LIN {X 0,Y 573.115,Z 294.058,A -85,B 0,C 180,E1 -2039.137,E2 -2039.137} C_VEL
LIN {X 0,Y 573.081,Z 298.172,A -85,B 0,C 180,E1 -2042.003,E2 -2042.003} C_VEL
LIN {X 0,Y 573.022,Z 301.873,A -85,B 0,C 180,E1 -2044.579,E2 -2044.579} C_VEL
LIN {X 0,Y 573.043,Z 305.517,A -85,B 0,C 180,E1 -2046.901,E2 -2046.901} C_VEL
LIN {X 0,Y 572.998,Z 309.134,A -85,B 0,C 180,E1 -2049.164,E2 -2049.164} C_VEL
LIN {X 0,Y 573.01,Z 312.764,A -85,B 0,C 180,E1 -2051.404,E2 -2051.404} C_VEL
LIN {X 0,Y 572.982,Z 314.48,A -85,B 0,C 180,E1 -2052.451,E2 -2052.451} C_VEL
LIN {X 0,Y 574.741,Z 322.312,A -85,B 0,C 180,E1 -2052.634,E2 -2052.634} C_VEL
LIN {X 0,Y 574.641,Z 337.953,A -85,B 0,C 180,E1 -2052.982,E2 -2052.982} C_VEL
LIN {X 0,Y 574.406,Z 353.082,A -85,B 0,C 180,E1 -2053.478,E2 -2053.478} C_VEL
LIN {X 0,Y 574.266,Z 365.728,A -85,B 0,C 180,E1 -2054.016,E2 -2054.016} C_VEL
LIN {X 0,Y 574.068,Z 377.863,A -85,B 0,C 180,E1 -2054.648,E2 -2054.648} C_VEL
LIN {X 0,Y 573.885,Z 391.295,A -85,B 0,C 180,E1 -2055.496,E2 -2055.496} C_VEL
LIN {X 0,Y 573.651,Z 404.761,A -85,B 0,C 180,E1 -2056.539,E2 -2056.539} C_VEL
LIN {X 0,Y 573.479,Z 416.274,A -85,B 0,C 180,E1 -2057.616,E2 -2057.616} C_VEL
LIN {X 0,Y 573.311,Z 426.306,A -85,B 0,C 180,E1 -2058.722,E2 -2058.722} C_VEL
LIN {X 0,Y 573.203,Z 436.788,A -85,B 0,C 180,E1 -2060.116,E2 -2060.116} C_VEL
LIN {X 0,Y 573.134,Z 444.469,A -85,B 0,C 180,E1 -2061.36,E2 -2061.36} C_VEL
LIN {X 0,Y 573.076,Z 450.883,A -85,B 0,C 180,E1 -2062.601,E2 -2062.601} C_VEL
LIN {X 0,Y 573.042,Z 456.782,A -85,B 0,C 180,E1 -2064.016,E2 -2064.016} C_VEL
LIN {X 0,Y 572.949,Z 460.255,A -85,B 0,C 180,E1 -2065.074,E2 -2065.074} C_VEL
LIN {X 0,Y 573.004,Z 463.808,A -85,B 0,C 180,E1 -2066.484,E2 -2066.484} C_VEL
LIN {X 0,Y 572.938,Z 466.135,A -85,B 0,C 180,E1 -2067.891,E2 -2067.891} C_VEL
LIN {X 0,Y 572.936,Z 467.306,A -85,B 0,C 180,E1 -2069.297,E2 -2069.297} C_VEL
LIN {X 0,Y 572.937,Z 467.337,A -85,B 0,C 180,E1 -2070.703,E2 -2070.703} C_VEL
LIN {X 0,Y 572.939,Z 466.235,A -85,B 0,C 180,E1 -2072.109,E2 -2072.109} C_VEL
LIN {X 0,Y 573.006,Z 463.992,A -85,B 0,C 180,E1 -2073.516,E2 -2073.516} C_VEL
LIN {X 0,Y 572.949,Z 460.527,A -85,B 0,C 180,E1 -2074.926,E2 -2074.926} C_VEL
LIN {X 0,Y 573.042,Z 457.098,A -85,B 0,C 180,E1 -2075.984,E2 -2075.984} C_VEL
LIN {X 0,Y 573.071,Z 451.302,A -85,B 0,C 180,E1 -2077.398,E2 -2077.398} C_VEL
LIN {X 0,Y 573.132,Z 444.977,A -85,B 0,C 180,E1 -2078.639,E2 -2078.639} C_VEL
LIN {X 0,Y 573.2,Z 437.38,A -85,B 0,C 180,E1 -2079.884,E2 -2079.884} C_VEL
LIN {X 0,Y 573.287,Z 428.365,A -85,B 0,C 180,E1 -2081.119,E2 -2081.119} C_VEL
LIN {X 0,Y 573.464,Z 417.166,A -85,B 0,C 180,E1 -2082.384,E2 -2082.384} C_VEL
LIN {X 0,Y 573.644,Z 406.815,A -85,B 0,C 180,E1 -2083.37,E2 -2083.37} C_VEL
LIN {X 0,Y 573.838,Z 395.714,A -85,B 0,C 180,E1 -2084.27,E2 -2084.27} C_VEL
LIN {X 0,Y 574.004,Z 382.508,A -85,B 0,C 180,E1 -2085.172,E2 -2085.172} C_VEL
LIN {X 0,Y 574.232,Z 369.513,A -85,B 0,C 180,E1 -2085.893,E2 -2085.893} C_VEL
LIN {X 0,Y 574.375,Z 356.387,A -85,B 0,C 180,E1 -2086.482,E2 -2086.482} C_VEL
LIN {X 0,Y 574.554,Z 342.236,A -85,B 0,C 180,E1 -2086.98,E2 -2086.98} C_VEL
LIN {X 0,Y 574.717,Z 327.066,A -85,B 0,C 180,E1 -2087.368,E2 -2087.368} C_VEL
LIN {X 0,Y 574.563,Z 321.22,A -85,B 0,C 180,E1 -2087.48,E2 -2087.48} C_VEL
LIN {X 0,Y 572.988,Z 314.455,A -85,B 0,C 180,E1 -2087.654,E2 -2087.654} C_VEL
LIN {X 0,Y 572.994,Z 310.49,A -85,B 0,C 180,E1 -2090.086,E2 -2090.086} C_VEL
LIN {X 0,Y 573.008,Z 306.857,A -85,B 0,C 180,E1 -2092.347,E2 -2092.347} C_VEL
LIN {X 0,Y 573.025,Z 302.942,A -85,B 0,C 180,E1 -2094.825,E2 -2094.825} C_VEL
LIN {X 0,Y 573.07,Z 299.762,A -85,B 0,C 180,E1 -2096.985,E2 -2096.985} C_VEL
LIN {X 0,Y 573.105,Z 296.219,A -85,B 0,C 180,E1 -2099.463,E2 -2099.463} C_VEL
LIN {X 0,Y 573.144,Z 292.244,A -85,B 0,C 180,E1 -2102.211,E2 -2102.211} C_VEL
LIN {X 0,Y 573.162,Z 287.996,A -85,B 0,C 180,E1 -2105.191,E2 -2105.191} C_VEL
LIN {X 0,Y 573.212,Z 284.101,A -85,B 0,C 180,E1 -2107.809,E2 -2107.809} C_VEL
LIN {X 0,Y 573.201,Z 279.714,A -85,B 0,C 180,E1 -2110.529,E2 -2110.529} C_VEL
LIN {X 0,Y 573.239,Z 279.706,A -85,B 0,C 180,E1 -2113.359,E2 -2113.359} C_VEL
LIN {X 0,Y 573.24,Z 279.703,A -85,B 0,C 180,E1 -2116.332,E2 -2116.332} C_VEL
LIN {X 0,Y 573.228,Z 279.71,A -85,B 0,C 180,E1 -2118.543,E2 -2118.543} C_VEL
LIN {X 0,Y 573.23,Z 279.703,A -85,B 0,C 180,E1 -2121.297,E2 -2121.297} C_VEL
LIN {X 0,Y 573.22,Z 279.707,A -85,B 0,C 180,E1 -2124.018,E2 -2124.018} C_VEL
LIN {X 0,Y 573.27,Z 279.7,A -85,B 0,C 180,E1 -2126.518,E2 -2126.518} C_VEL
LIN {X 0,Y 573.226,Z 279.704,A -85,B 0,C 180,E1 -2129.118,E2 -2129.118} C_VEL
LIN {X 0,Y 573.194,Z 279.714,A -85,B 0,C 180,E1 -2131.982,E2 -2131.982} C_VEL
LIN {X 0,Y 573.238,Z 279.701,A -85,B 0,C 180,E1 -2134.589,E2 -2134.589} C_VEL
LIN {X 0,Y 573.236,Z 279.701,A -85,B 0,C 180,E1 -2137.662,E2 -2137.662} C_VEL
LIN {X 0,Y 573.267,Z 279.701,A -85,B 0,C 180,E1 -2140.67,E2 -2140.67} C_VEL
LIN {X 0,Y 573.221,Z 279.709,A -85,B 0,C 180,E1 -2143.621,E2 -2143.621} C_VEL
LIN {X 0,Y 573.273,Z 279.699,A -85,B 0,C 180,E1 -2145.807,E2 -2145.807} C_VEL
LIN {X 0,Y 573.264,Z 279.703,A -85,B 0,C 180,E1 -2148.745,E2 -2148.745} C_VEL
LIN {X 0,Y 573.252,Z 279.703,A -85,B 0,C 180,E1 -2151.54,E2 -2151.54} C_VEL
LIN {X 0,Y 573.262,Z 279.697,A -85,B 0,C 180,E1 -2154.371,E2 -2154.371} C_VEL
LIN {X 0,Y 573.309,Z 279.697,A -85,B 0,C 180,E1 -2157.189,E2 -2157.189} C_VEL
LIN {X 0,Y 573.324,Z 279.693,A -85,B 0,C 180,E1 -2160,E2 -2160} C_VEL
LIN {X 0,Y 573.287,Z 279.696,A -85,B 0,C 180,E1 -2162.811,E2 -2162.811} C_VEL
LIN {X 0,Y 573.28,Z 279.698,A -85,B 0,C 180,E1 -2165.628,E2 -2165.628} C_VEL
LIN {X 0,Y 573.255,Z 279.706,A -85,B 0,C 180,E1 -2168.46,E2 -2168.46} C_VEL
LIN {X 0,Y 573.273,Z 279.696,A -85,B 0,C 180,E1 -2171.312,E2 -2171.312} C_VEL
LIN {X 0,Y 573.244,Z 279.701,A -85,B 0,C 180,E1 -2174.409,E2 -2174.409} C_VEL
LIN {X 0,Y 573.247,Z 279.705,A -85,B 0,C 180,E1 -2177.112,E2 -2177.112} C_VEL
LIN {X 0,Y 573.253,Z 279.705,A -85,B 0,C 180,E1 -2180.077,E2 -2180.077} C_VEL
LIN {X 0,Y 573.235,Z 279.703,A -85,B 0,C 180,E1 -2183.099,E2 -2183.099} C_VEL
LIN {X 0,Y 573.233,Z 279.702,A -85,B 0,C 180,E1 -2186.191,E2 -2186.191} C_VEL
LIN {X 0,Y 573.229,Z 279.71,A -85,B 0,C 180,E1 -2188.565,E2 -2188.565} C_VEL
LIN {X 0,Y 573.23,Z 279.703,A -85,B 0,C 180,E1 -2190.993,E2 -2190.993} C_VEL
LIN {X 0,Y 573.263,Z 279.706,A -85,B 0,C 180,E1 -2193.524,E2 -2193.524} C_VEL
LIN {X 0,Y 573.19,Z 279.708,A -85,B 0,C 180,E1 -2196.053,E2 -2196.053} C_VEL
LIN {X 0,Y 573.232,Z 279.708,A -85,B 0,C 180,E1 -2198.702,E2 -2198.702} C_VEL
LIN {X 0,Y 573.237,Z 279.706,A -85,B 0,C 180,E1 -2201.594,E2 -2201.594} C_VEL
LIN {X 0,Y 573.225,Z 279.703,A -85,B 0,C 180,E1 -2204.334,E2 -2204.334} C_VEL
LIN {X 0,Y 573.218,Z 279.706,A -85,B 0,C 180,E1 -2207.361,E2 -2207.361} C_VEL
LIN {X 0,Y 573.236,Z 279.709,A -85,B 0,C 180,E1 -2210.392,E2 -2210.392} C_VEL
LIN {X 0,Y 573.252,Z 279.707,A -85,B 0,C 180,E1 -2213.078,E2 -2213.078} C_VEL
LIN {X 0,Y 573.217,Z 279.814,A -85,B 0,C 180,E1 -2214.166,E2 -2214.166} C_VEL
LIN {X 0,Y 575.333,Z 288.451,A -85,B 0,C 180,E1 -2215.812,E2 -2215.812} C_VEL
LIN {X 0,Y 574.902,Z 304.368,A -85,B 0,C 180,E1 -2218.459,E2 -2218.459} C_VEL
LIN {X 0,Y 574.675,Z 320.037,A -85,B 0,C 180,E1 -2220.914,E2 -2220.914} C_VEL
LIN {X 0,Y 574.403,Z 337.41,A -85,B 0,C 180,E1 -2223.567,E2 -2223.567} C_VEL
LIN {X 0,Y 574.164,Z 354.72,A -85,B 0,C 180,E1 -2226.176,E2 -2226.176} C_VEL
LIN {X 0,Y 573.88,Z 375.193,A -85,B 0,C 180,E1 -2229.198,E2 -2229.198} C_VEL
LIN {X 0,Y 573.658,Z 394.386,A -85,B 0,C 180,E1 -2231.98,E2 -2231.98} C_VEL
LIN {X 0,Y 573.656,Z 396.802,A -85,B 0,C 180,E1 -2232.329,E2 -2232.329} C_VEL
LIN {X 0,Y 574.768,Z 403.436,A -85,B 0,C 180,E1 -2232.451,E2 -2232.451} C_VEL
LIN {X 0,Y 574.667,Z 419.595,A -85,B 0,C 180,E1 -2232.729,E2 -2232.729} C_VEL
LIN {X 0,Y 574.555,Z 435.297,A -85,B 0,C 180,E1 -2233.157,E2 -2233.157} C_VEL
LIN {X 0,Y 574.348,Z 449.799,A -85,B 0,C 180,E1 -2233.7,E2 -2233.7} C_VEL
LIN {X 0,Y 574.157,Z 463.874,A -85,B 0,C 180,E1 -2234.378,E2 -2234.378} C_VEL
LIN {X 0,Y 573.982,Z 476.044,A -85,B 0,C 180,E1 -2235.1,E2 -2235.1} C_VEL
LIN {X 0,Y 573.748,Z 488.699,A -85,B 0,C 180,E1 -2236,E2 -2236} C_VEL
LIN {X 0,Y 573.581,Z 499.336,A -85,B 0,C 180,E1 -2236.899,E2 -2236.899} C_VEL
LIN {X 0,Y 573.405,Z 510.141,A -85,B 0,C 180,E1 -2237.974,E2 -2237.974} C_VEL
LIN {X 0,Y 573.3,Z 519.79,A -85,B 0,C 180,E1 -2239.111,E2 -2239.111} C_VEL
LIN {X 0,Y 573.188,Z 528.295,A -85,B 0,C 180,E1 -2240.294,E2 -2240.294} C_VEL
LIN {X 0,Y 573.109,Z 535.751,A -85,B 0,C 180,E1 -2241.538,E2 -2241.538} C_VEL
LIN {X 0,Y 573.047,Z 542.702,A -85,B 0,C 180,E1 -2242.956,E2 -2242.956} C_VEL
LIN {X 0,Y 573.055,Z 548.161,A -85,B 0,C 180,E1 -2244.37,E2 -2244.37} C_VEL
LIN {X 0,Y 573.006,Z 552.29,A -85,B 0,C 180,E1 -2245.78,E2 -2245.78} C_VEL
LIN {X 0,Y 572.955,Z 555.188,A -85,B 0,C 180,E1 -2247.188,E2 -2247.188} C_VEL
LIN {X 0,Y 572.944,Z 556.912,A -85,B 0,C 180,E1 -2248.594,E2 -2248.594} C_VEL
LIN {X 0,Y 572.935,Z 557.5,A -85,B 0,C 180,E1 -2250,E2 -2250} C_VEL
LIN {X 0,Y 572.944,Z 556.911,A -85,B 0,C 180,E1 -2251.406,E2 -2251.406} C_VEL
LIN {X 0,Y 572.955,Z 555.186,A -85,B 0,C 180,E1 -2252.813,E2 -2252.813} C_VEL
LIN {X 0,Y 573.007,Z 552.288,A -85,B 0,C 180,E1 -2254.22,E2 -2254.22} C_VEL
LIN {X 0,Y 573.055,Z 548.162,A -85,B 0,C 180,E1 -2255.631,E2 -2255.631} C_VEL
LIN {X 0,Y 573.048,Z 542.701,A -85,B 0,C 180,E1 -2257.045,E2 -2257.045} C_VEL
LIN {X 0,Y 573.109,Z 535.748,A -85,B 0,C 180,E1 -2258.462,E2 -2258.462} C_VEL
LIN {X 0,Y 573.199,Z 527.087,A -85,B 0,C 180,E1 -2259.884,E2 -2259.884} C_VEL
LIN {X 0,Y 573.295,Z 517.948,A -85,B 0,C 180,E1 -2261.124,E2 -2261.124} C_VEL
LIN {X 0,Y 573.453,Z 508.507,A -85,B 0,C 180,E1 -2262.205,E2 -2262.205} C_VEL
LIN {X 0,Y 573.628,Z 497.383,A -85,B 0,C 180,E1 -2263.281,E2 -2263.281} C_VEL
LIN {X 0,Y 573.828,Z 485.135,A -85,B 0,C 180,E1 -2264.274,E2 -2264.274} C_VEL
LIN {X 0,Y 574.016,Z 471.775,A -85,B 0,C 180,E1 -2265.172,E2 -2265.172} C_VEL
LIN {X 0,Y 574.222,Z 458.597,A -85,B 0,C 180,E1 -2265.894,E2 -2265.894} C_VEL
LIN {X 0,Y 574.416,Z 444.173,A -85,B 0,C 180,E1 -2266.527,E2 -2266.527} C_VEL
LIN {X 0,Y 574.592,Z 429.245,A -85,B 0,C 180,E1 -2267.025,E2 -2267.025} C_VEL
LIN {X 0,Y 574.68,Z 414.321,A -85,B 0,C 180,E1 -2267.377,E2 -2267.377} C_VEL
LIN {X 0,Y 574.609,Z 401.989,A -85,B 0,C 180,E1 -2267.572,E2 -2267.572} C_VEL
LIN {X 0,Y 573.643,Z 396.706,A -85,B 0,C 180,E1 -2267.686,E2 -2267.686} C_VEL
LIN {X 0,Y 573.874,Z 377.749,A -85,B 0,C 180,E1 -2270.428,E2 -2270.428} C_VEL
LIN {X 0,Y 574.128,Z 357.888,A -85,B 0,C 180,E1 -2273.352,E2 -2273.352} C_VEL
LIN {X 0,Y 574.401,Z 339.363,A -85,B 0,C 180,E1 -2276.134,E2 -2276.134} C_VEL
LIN {X 0,Y 574.615,Z 323.851,A -85,B 0,C 180,E1 -2278.49,E2 -2278.49} C_VEL
LIN {X 0,Y 574.762,Z 310.765,A -85,B 0,C 180,E1 -2280.494,E2 -2280.494} C_VEL
LIN {X 0,Y 575.281,Z 296.37,A -85,B 0,C 180,E1 -2282.932,E2 -2282.932} C_VEL
LIN {X 0,Y 575.707,Z 289.67,A -85,B 0,C 180,E1 -2284.163,E2 -2284.163} C_VEL
LIN {X 0,Y 574.296,Z 283.704,A -85,B 0,C 180,E1 -2285.541,E2 -2285.541} C_VEL
LIN {X 0,Y 573.22,Z 279.71,A -85,B 0,C 180,E1 -2286.651,E2 -2286.651} C_VEL
LIN {X 0,Y 573.247,Z 279.707,A -85,B 0,C 180,E1 -2289.607,E2 -2289.607} C_VEL
LIN {X 0,Y 573.245,Z 279.708,A -85,B 0,C 180,E1 -2292.642,E2 -2292.642} C_VEL
LIN {X 0,Y 573.224,Z 279.709,A -85,B 0,C 180,E1 -2295.665,E2 -2295.665} C_VEL
LIN {X 0,Y 573.234,Z 279.707,A -85,B 0,C 180,E1 -2298.543,E2 -2298.543} C_VEL
LIN {X 0,Y 573.245,Z 279.706,A -85,B 0,C 180,E1 -2301.299,E2 -2301.299} C_VEL
LIN {X 0,Y 573.189,Z 279.715,A -85,B 0,C 180,E1 -2304.022,E2 -2304.022} C_VEL
LIN {X 0,Y 573.289,Z 282.484,A -85,B 0,C 180,E1 -2306.519,E2 -2306.519} C_VEL
LIN {X 0,Y 573.241,Z 285.279,A -85,B 0,C 180,E1 -2309.116,E2 -2309.116} C_VEL
LIN {X 0,Y 573.262,Z 287.554,A -85,B 0,C 180,E1 -2311.437,E2 -2311.437} C_VEL
LIN {X 0,Y 573.201,Z 289.676,A -85,B 0,C 180,E1 -2313.807,E2 -2313.807} C_VEL
LIN {X 0,Y 573.084,Z 291.517,A -85,B 0,C 180,E1 -2316.128,E2 -2316.128} C_VEL
LIN {X 0,Y 572.988,Z 294.122,A -85,B 0,C 180,E1 -2319.164,E2 -2319.164} C_VEL
LIN {X 0,Y 572.965,Z 296.701,A -85,B 0,C 180,E1 -2321.403,E2 -2321.403} C_VEL
LIN {X 0,Y 572.967,Z 299.405,A -85,B 0,C 180,E1 -2323.613,E2 -2323.613} C_VEL
LIN {X 0,Y 572.986,Z 303.009,A -85,B 0,C 180,E1 -2326.524,E2 -2326.524} C_VEL
LIN {X 0,Y 572.999,Z 304.333,A -85,B 0,C 180,E1 -2327.583,E2 -2327.583} C_VEL
LIN {X 0,Y 573.818,Z 310.855,A -85,B 0,C 180,E1 -2327.758,E2 -2327.758} C_VEL
LIN {X 0,Y 573.71,Z 324.273,A -85,B 0,C 180,E1 -2328.16,E2 -2328.16} C_VEL
LIN {X 0,Y 573.629,Z 336.787,A -85,B 0,C 180,E1 -2328.695,E2 -2328.695} C_VEL
LIN {X 0,Y 573.528,Z 347.998,A -85,B 0,C 180,E1 -2329.321,E2 -2329.321} C_VEL
LIN {X 0,Y 573.35,Z 359.337,A -85,B 0,C 180,E1 -2330.119,E2 -2330.119} C_VEL
LIN {X 0,Y 573.28,Z 369.385,A -85,B 0,C 180,E1 -2331.008,E2 -2331.008} C_VEL
LIN {X 0,Y 573.161,Z 379.087,A -85,B 0,C 180,E1 -2332.071,E2 -2332.071} C_VEL
LIN {X 0,Y 573.093,Z 387.022,A -85,B 0,C 180,E1 -2333.163,E2 -2333.163} C_VEL
LIN {X 0,Y 573.07,Z 393.948,A -85,B 0,C 180,E1 -2334.37,E2 -2334.37} C_VEL
LIN {X 0,Y 573.029,Z 398.691,A -85,B 0,C 180,E1 -2335.428,E2 -2335.428} C_VEL
LIN {X 0,Y 573.023,Z 402.323,A -85,B 0,C 180,E1 -2336.484,E2 -2336.484} C_VEL
LIN {X 0,Y 572.959,Z 404.2,A -85,B 0,C 180,E1 -2337.188,E2 -2337.188} C_VEL
LIN {X 0,Y 572.938,Z 405.627,A -85,B 0,C 180,E1 -2337.891,E2 -2337.891} C_VEL
LIN {X 0,Y 572.942,Z 407.255,A -85,B 0,C 180,E1 -2339.297,E2 -2339.297} C_VEL
LIN {X 0,Y 572.938,Z 407.496,A -85,B 0,C 180,E1 -2340,E2 -2340} C_VEL
LIN {X 0,Y 572.941,Z 407.315,A -85,B 0,C 180,E1 -2340.703,E2 -2340.703} C_VEL
LIN {X 0,Y 572.937,Z 405.772,A -85,B 0,C 180,E1 -2342.109,E2 -2342.109} C_VEL
LIN {X 0,Y 572.96,Z 404.411,A -85,B 0,C 180,E1 -2342.812,E2 -2342.812} C_VEL
LIN {X 0,Y 573.015,Z 401.532,A -85,B 0,C 180,E1 -2343.868,E2 -2343.868} C_VEL
LIN {X 0,Y 572.963,Z 397.631,A -85,B 0,C 180,E1 -2344.926,E2 -2344.926} C_VEL
LIN {X 0,Y 573.075,Z 392.601,A -85,B 0,C 180,E1 -2345.984,E2 -2345.984} C_VEL
LIN {X 0,Y 573.083,Z 386.275,A -85,B 0,C 180,E1 -2347.044,E2 -2347.044} C_VEL
LIN {X 0,Y 573.175,Z 378.354,A -85,B 0,C 180,E1 -2348.106,E2 -2348.106} C_VEL
LIN {X 0,Y 573.287,Z 368.504,A -85,B 0,C 180,E1 -2349.17,E2 -2349.17} C_VEL
LIN {X 0,Y 573.416,Z 358.18,A -85,B 0,C 180,E1 -2350.059,E2 -2350.059} C_VEL
LIN {X 0,Y 573.544,Z 346.593,A -85,B 0,C 180,E1 -2350.856,E2 -2350.856} C_VEL
LIN {X 0,Y 573.658,Z 335.698,A -85,B 0,C 180,E1 -2351.449,E2 -2351.449} C_VEL
LIN {X 0,Y 573.718,Z 324.526,A -85,B 0,C 180,E1 -2351.921,E2 -2351.921} C_VEL
LIN {X 0,Y 573.827,Z 311.765,A -85,B 0,C 180,E1 -2352.309,E2 -2352.309} C_VEL
LIN {X 0,Y 573.379,Z 307.024,A -85,B 0,C 180,E1 -2352.428,E2 -2352.428} C_VEL
LIN {X 0,Y 572.963,Z 304.333,A -85,B 0,C 180,E1 -2352.508,E2 -2352.508} C_VEL
LIN {X 0,Y 572.959,Z 301.318,A -85,B 0,C 180,E1 -2354.927,E2 -2354.927} C_VEL
LIN {X 0,Y 572.943,Z 298.246,A -85,B 0,C 180,E1 -2357.422,E2 -2357.422} C_VEL
LIN {X 0,Y 572.979,Z 295.007,A -85,B 0,C 180,E1 -2360.087,E2 -2360.087} C_VEL
LIN {X 0,Y 572.968,Z 294.558,A -85,B 0,C 180,E1 -2360.463,E2 -2360.463} C_VEL
LIN {X 0,Y 572.312,Z 293.943,A -85,B 0,C 180,E1 -2361.046,E2 -2361.046} C_VEL
LIN {X 0,Y 569.466,Z 293.15,A -85,B 0,C 180,E1 -2361.995,E2 -2361.995} C_VEL
LIN {X 0,Y 567.052,Z 292.543,A -85,B 0,C 180,E1 -2362.759,E2 -2362.759} C_VEL
LIN {X 0,Y 566.01,Z 292.015,A -85,B 0,C 180,E1 -2363.348,E2 -2363.348} C_VEL
LIN {X 0,Y 565.923,Z 291.817,A -85,B 0,C 180,E1 -2363.547,E2 -2363.547} C_VEL
LIN {X 0,Y 565.974,Z 289.57,A -85,B 0,C 180,E1 -2365.761,E2 -2365.761} C_VEL
LIN {X 0,Y 566.002,Z 286.959,A -85,B 0,C 180,E1 -2368.163,E2 -2368.163} C_VEL
LIN {X 0,Y 565.98,Z 284.379,A -85,B 0,C 180,E1 -2370.605,E2 -2370.605} C_VEL
LIN {X 0,Y 565.98,Z 281.51,A -85,B 0,C 180,E1 -2373.118,E2 -2373.118} C_VEL
LIN {X 0,Y 566.008,Z 280.61,A -85,B 0,C 180,E1 -2373.97,E2 -2373.97} C_VEL
LIN {X 0,Y 566.194,Z 280.58,A -85,B 0,C 180,E1 -2376.57,E2 -2376.57} C_VEL
LIN {X 0,Y 566.225,Z 280.575,A -85,B 0,C 180,E1 -2379.687,E2 -2379.687} C_VEL
LIN {X 0,Y 566.203,Z 280.58,A -85,B 0,C 180,E1 -2382.917,E2 -2382.917} C_VEL
LIN {X 0,Y 566.161,Z 280.588,A -85,B 0,C 180,E1 -2385.96,E2 -2385.96} C_VEL
LIN {X 0,Y 566.168,Z 280.589,A -85,B 0,C 180,E1 -2388.142,E2 -2388.142} C_VEL
LIN {X 0,Y 566.136,Z 280.74,A -85,B 0,C 180,E1 -2389.794,E2 -2389.794} C_VEL
LIN {X 0,Y 566.165,Z 285.409,A -85,B 0,C 180,E1 -2392.604,E2 -2392.604} C_VEL
LIN {X 0,Y 566.113,Z 289.214,A -85,B 0,C 180,E1 -2395.175,E2 -2395.175} C_VEL
LIN {X 0,Y 566.091,Z 292.826,A -85,B 0,C 180,E1 -2397.734,E2 -2397.734} C_VEL
LIN {X 0,Y 566.052,Z 296.586,A -85,B 0,C 180,E1 -2400.355,E2 -2400.355} C_VEL
LIN {X 0,Y 566.001,Z 299.877,A -85,B 0,C 180,E1 -2402.65,E2 -2402.65} C_VEL
LIN {X 0,Y 565.963,Z 303.211,A -85,B 0,C 180,E1 -2405.026,E2 -2405.026} C_VEL
LIN {X 0,Y 565.948,Z 306.714,A -85,B 0,C 180,E1 -2407.358,E2 -2407.358} C_VEL
LIN {X 0,Y 565.931,Z 311.555,A -85,B 0,C 180,E1 -2410.409,E2 -2410.409} C_VEL
LIN {X 0,Y 565.893,Z 314.463,A -85,B 0,C 180,E1 -2412.213,E2 -2412.213} C_VEL
LIN {X 0,Y 567.959,Z 323.511,A -85,B 0,C 180,E1 -2412.44,E2 -2412.44} C_VEL
LIN {X 0,Y 567.805,Z 340.105,A -85,B 0,C 180,E1 -2412.836,E2 -2412.836} C_VEL
LIN {X 0,Y 567.57,Z 353.381,A -85,B 0,C 180,E1 -2413.285,E2 -2413.285} C_VEL
LIN {X 0,Y 567.408,Z 365.723,A -85,B 0,C 180,E1 -2413.818,E2 -2413.818} C_VEL
LIN {X 0,Y 567.203,Z 377.86,A -85,B 0,C 180,E1 -2414.458,E2 -2414.458} C_VEL
LIN {X 0,Y 567,Z 390.624,A -85,B 0,C 180,E1 -2415.268,E2 -2415.268} C_VEL
LIN {X 0,Y 566.727,Z 403.712,A -85,B 0,C 180,E1 -2416.28,E2 -2416.28} C_VEL
LIN {X 0,Y 566.535,Z 414.488,A -85,B 0,C 180,E1 -2417.279,E2 -2417.279} C_VEL
LIN {X 0,Y 566.338,Z 424.498,A -85,B 0,C 180,E1 -2418.366,E2 -2418.366} C_VEL
LIN {X 0,Y 566.226,Z 434.328,A -85,B 0,C 180,E1 -2419.632,E2 -2419.632} C_VEL
LIN {X 0,Y 566.057,Z 443.461,A -85,B 0,C 180,E1 -2421.072,E2 -2421.072} C_VEL
LIN {X 0,Y 566.016,Z 449.187,A -85,B 0,C 180,E1 -2422.15,E2 -2422.15} C_VEL
LIN {X 0,Y 565.946,Z 454.844,A -85,B 0,C 180,E1 -2423.44,E2 -2423.44} C_VEL
LIN {X 0,Y 565.926,Z 459.16,A -85,B 0,C 180,E1 -2424.656,E2 -2424.656} C_VEL
LIN {X 0,Y 565.913,Z 462.163,A -85,B 0,C 180,E1 -2425.727,E2 -2425.727} C_VEL
LIN {X 0,Y 565.872,Z 465.109,A -85,B 0,C 180,E1 -2427.152,E2 -2427.152} C_VEL
LIN {X 0,Y 565.842,Z 466.88,A -85,B 0,C 180,E1 -2428.576,E2 -2428.576} C_VEL
LIN {X 0,Y 565.837,Z 467.496,A -85,B 0,C 180,E1 -2430,E2 -2430} C_VEL
LIN {X 0,Y 565.844,Z 466.959,A -85,B 0,C 180,E1 -2431.423,E2 -2431.423} C_VEL
LIN {X 0,Y 565.874,Z 465.262,A -85,B 0,C 180,E1 -2432.847,E2 -2432.847} C_VEL
LIN {X 0,Y 565.913,Z 462.382,A -85,B 0,C 180,E1 -2434.273,E2 -2434.273} C_VEL
LIN {X 0,Y 565.982,Z 458.318,A -85,B 0,C 180,E1 -2435.701,E2 -2435.701} C_VEL
LIN {X 0,Y 565.974,Z 452.914,A -85,B 0,C 180,E1 -2437.133,E2 -2437.133} C_VEL
LIN {X 0,Y 566.058,Z 445.968,A -85,B 0,C 180,E1 -2438.568,E2 -2438.568} C_VEL
LIN {X 0,Y 566.125,Z 438.535,A -85,B 0,C 180,E1 -2439.828,E2 -2439.828} C_VEL
LIN {X 0,Y 566.253,Z 430.628,A -85,B 0,C 180,E1 -2440.956,E2 -2440.956} C_VEL
LIN {X 0,Y 566.415,Z 420.564,A -85,B 0,C 180,E1 -2442.177,E2 -2442.177} C_VEL
LIN {X 0,Y 566.627,Z 408.849,A -85,B 0,C 180,E1 -2443.356,E2 -2443.356} C_VEL
LIN {X 0,Y 566.833,Z 398.076,A -85,B 0,C 180,E1 -2444.266,E2 -2444.266} C_VEL
LIN {X 0,Y 567.092,Z 386.68,A -85,B 0,C 180,E1 -2445.085,E2 -2445.085} C_VEL
LIN {X 0,Y 567.267,Z 374.623,A -85,B 0,C 180,E1 -2445.817,E2 -2445.817} C_VEL
LIN {X 0,Y 567.486,Z 359.752,A -85,B 0,C 180,E1 -2446.549,E2 -2446.549} C_VEL
LIN {X 0,Y 567.734,Z 345.452,A -85,B 0,C 180,E1 -2447.086,E2 -2447.086} C_VEL
LIN {X 0,Y 567.872,Z 332.079,A -85,B 0,C 180,E1 -2447.465,E2 -2447.465} C_VEL
LIN {X 0,Y 567.817,Z 322.587,A -85,B 0,C 180,E1 -2447.67,E2 -2447.67} C_VEL
LIN {X 0,Y 565.89,Z 314.454,A -85,B 0,C 180,E1 -2447.883,E2 -2447.883} C_VEL
LIN {X 0,Y 565.897,Z 310.489,A -85,B 0,C 180,E1 -2450.349,E2 -2450.349} C_VEL
LIN {X 0,Y 565.944,Z 305.937,A -85,B 0,C 180,E1 -2453.227,E2 -2453.227} C_VEL
LIN {X 0,Y 565.978,Z 302.22,A -85,B 0,C 180,E1 -2455.76,E2 -2455.76} C_VEL
LIN {X 0,Y 566.064,Z 298.826,A -85,B 0,C 180,E1 -2458.175,E2 -2458.175} C_VEL
LIN {X 0,Y 566.076,Z 294.69,A -85,B 0,C 180,E1 -2461.057,E2 -2461.057} C_VEL
LIN {X 0,Y 566.08,Z 290.554,A -85,B 0,C 180,E1 -2463.965,E2 -2463.965} C_VEL
LIN {X 0,Y 566.136,Z 286.808,A -85,B 0,C 180,E1 -2466.575,E2 -2466.575} C_VEL
LIN {X 0,Y 566.164,Z 282.514,A -85,B 0,C 180,E1 -2469.278,E2 -2469.278} C_VEL
LIN {X 0,Y 566.135,Z 280.896,A -85,B 0,C 180,E1 -2470.205,E2 -2470.205} C_VEL
LIN {X 0,Y 566.14,Z 280.59,A -85,B 0,C 180,E1 -2471.143,E2 -2471.143} C_VEL
LIN {X 0,Y 566.197,Z 280.582,A -85,B 0,C 180,E1 -2474.036,E2 -2474.036} C_VEL
LIN {X 0,Y 566.202,Z 280.585,A -85,B 0,C 180,E1 -2477.083,E2 -2477.083} C_VEL
LIN {X 0,Y 566.205,Z 280.58,A -85,B 0,C 180,E1 -2479.801,E2 -2479.801} C_VEL
LIN {X 0,Y 566.188,Z 280.581,A -85,B 0,C 180,E1 -2482.601,E2 -2482.601} C_VEL
LIN {X 0,Y 566.211,Z 280.584,A -85,B 0,C 180,E1 -2485.182,E2 -2485.182} C_VEL
LIN {X 0,Y 566.23,Z 280.576,A -85,B 0,C 180,E1 -2487.743,E2 -2487.743} C_VEL
LIN {X 0,Y 566.167,Z 280.589,A -85,B 0,C 180,E1 -2490.335,E2 -2490.335} C_VEL
LIN {X 0,Y 566.178,Z 280.586,A -85,B 0,C 180,E1 -2493.457,E2 -2493.457} C_VEL
LIN {X 0,Y 566.197,Z 280.581,A -85,B 0,C 180,E1 -2495.819,E2 -2495.819} C_VEL
LIN {X 0,Y 566.209,Z 280.58,A -85,B 0,C 180,E1 -2498.902,E2 -2498.902} C_VEL
LIN {X 0,Y 566.188,Z 280.581,A -85,B 0,C 180,E1 -2501.172,E2 -2501.172} C_VEL
LIN {X 0,Y 566.184,Z 280.581,A -85,B 0,C 180,E1 -2504.152,E2 -2504.152} C_VEL
LIN {X 0,Y 566.197,Z 280.58,A -85,B 0,C 180,E1 -2506.359,E2 -2506.359} C_VEL
LIN {X 0,Y 566.236,Z 280.579,A -85,B 0,C 180,E1 -2508.675,E2 -2508.675} C_VEL
LIN {X 0,Y 566.203,Z 280.58,A -85,B 0,C 180,E1 -2511.434,E2 -2511.434} C_VEL
LIN {X 0,Y 566.231,Z 280.573,A -85,B 0,C 180,E1 -2514.301,E2 -2514.301} C_VEL
LIN {X 0,Y 566.274,Z 280.573,A -85,B 0,C 180,E1 -2517.154,E2 -2517.154} C_VEL
LIN {X 0,Y 566.294,Z 280.568,A -85,B 0,C 180,E1 -2520,E2 -2520} C_VEL
LIN {X 0,Y 566.255,Z 280.572,A -85,B 0,C 180,E1 -2522.846,E2 -2522.846} C_VEL
LIN {X 0,Y 566.246,Z 280.573,A -85,B 0,C 180,E1 -2525.698,E2 -2525.698} C_VEL
LIN {X 0,Y 566.208,Z 280.585,A -85,B 0,C 180,E1 -2528.566,E2 -2528.566} C_VEL
LIN {X 0,Y 566.243,Z 280.572,A -85,B 0,C 180,E1 -2531.454,E2 -2531.454} C_VEL
LIN {X 0,Y 566.202,Z 280.579,A -85,B 0,C 180,E1 -2534.493,E2 -2534.493} C_VEL
LIN {X 0,Y 566.189,Z 280.581,A -85,B 0,C 180,E1 -2537.332,E2 -2537.332} C_VEL
LIN {X 0,Y 566.214,Z 280.581,A -85,B 0,C 180,E1 -2540.337,E2 -2540.337} C_VEL
LIN {X 0,Y 566.167,Z 280.585,A -85,B 0,C 180,E1 -2543.28,E2 -2543.28} C_VEL
LIN {X 0,Y 566.186,Z 280.58,A -85,B 0,C 180,E1 -2545.75,E2 -2545.75} C_VEL
LIN {X 0,Y 566.184,Z 280.583,A -85,B 0,C 180,E1 -2548.198,E2 -2548.198} C_VEL
LIN {X 0,Y 566.195,Z 280.58,A -85,B 0,C 180,E1 -2551.077,E2 -2551.077} C_VEL
LIN {X 0,Y 566.212,Z 280.582,A -85,B 0,C 180,E1 -2553.734,E2 -2553.734} C_VEL
LIN {X 0,Y 566.176,Z 280.585,A -85,B 0,C 180,E1 -2556.572,E2 -2556.572} C_VEL
LIN {X 0,Y 566.211,Z 280.579,A -85,B 0,C 180,E1 -2559.685,E2 -2559.685} C_VEL
LIN {X 0,Y 566.209,Z 280.582,A -85,B 0,C 180,E1 -2562.088,E2 -2562.088} C_VEL
LIN {X 0,Y 566.167,Z 280.587,A -85,B 0,C 180,E1 -2565.036,E2 -2565.036} C_VEL
LIN {X 0,Y 566.169,Z 280.583,A -85,B 0,C 180,E1 -2567.909,E2 -2567.909} C_VEL
LIN {X 0,Y 566.213,Z 280.581,A -85,B 0,C 180,E1 -2570.726,E2 -2570.726} C_VEL
LIN {X 0,Y 566.175,Z 280.601,A -85,B 0,C 180,E1 -2573.769,E2 -2573.769} C_VEL
LIN {X 0,Y 568.189,Z 288.461,A -85,B 0,C 180,E1 -2575.321,E2 -2575.321} C_VEL
LIN {X 0,Y 568.595,Z 291.68,A -85,B 0,C 180,E1 -2575.908,E2 -2575.908} C_VEL
LIN {X 0,Y 568.116,Z 308.29,A -85,B 0,C 180,E1 -2578.697,E2 -2578.697} C_VEL
LIN {X 0,Y 567.765,Z 326.881,A -85,B 0,C 180,E1 -2581.619,E2 -2581.619} C_VEL
LIN {X 0,Y 567.457,Z 346.171,A -85,B 0,C 180,E1 -2584.571,E2 -2584.571} C_VEL
LIN {X 0,Y 567.117,Z 363.677,A -85,B 0,C 180,E1 -2587.216,E2 -2587.216} C_VEL
LIN {X 0,Y 566.886,Z 382.87,A -85,B 0,C 180,E1 -2590.066,E2 -2590.066} C_VEL
LIN {X 0,Y 566.677,Z 396.818,A -85,B 0,C 180,E1 -2592.106,E2 -2592.106} C_VEL
LIN {X 0,Y 567.96,Z 403.517,A -85,B 0,C 180,E1 -2592.235,E2 -2592.235} C_VEL
LIN {X 0,Y 567.889,Z 419.351,A -85,B 0,C 180,E1 -2592.511,E2 -2592.511} C_VEL
LIN {X 0,Y 567.739,Z 435.296,A -85,B 0,C 180,E1 -2592.949,E2 -2592.949} C_VEL
LIN {X 0,Y 567.519,Z 449.8,A -85,B 0,C 180,E1 -2593.498,E2 -2593.498} C_VEL
LIN {X 0,Y 567.289,Z 463.877,A -85,B 0,C 180,E1 -2594.184,E2 -2594.184} C_VEL
LIN {X 0,Y 567.073,Z 477.18,A -85,B 0,C 180,E1 -2594.988,E2 -2594.988} C_VEL
LIN {X 0,Y 566.8,Z 489.861,A -85,B 0,C 180,E1 -2595.916,E2 -2595.916} C_VEL
LIN {X 0,Y 566.577,Z 501.278,A -85,B 0,C 180,E1 -2596.916,E2 -2596.916} C_VEL
LIN {X 0,Y 566.371,Z 511.767,A -85,B 0,C 180,E1 -2598.004,E2 -2598.004} C_VEL
LIN {X 0,Y 566.275,Z 520.362,A -85,B 0,C 180,E1 -2599.05,E2 -2599.05} C_VEL
LIN {X 0,Y 566.123,Z 529.417,A -85,B 0,C 180,E1 -2600.352,E2 -2600.352} C_VEL
LIN {X 0,Y 566.061,Z 535.751,A -85,B 0,C 180,E1 -2601.432,E2 -2601.432} C_VEL
LIN {X 0,Y 565.974,Z 542.702,A -85,B 0,C 180,E1 -2602.867,E2 -2602.867} C_VEL
LIN {X 0,Y 565.982,Z 548.161,A -85,B 0,C 180,E1 -2604.299,E2 -2604.299} C_VEL
LIN {X 0,Y 565.912,Z 552.29,A -85,B 0,C 180,E1 -2605.727,E2 -2605.727} C_VEL
LIN {X 0,Y 565.873,Z 555.187,A -85,B 0,C 180,E1 -2607.153,E2 -2607.153} C_VEL
LIN {X 0,Y 565.844,Z 556.911,A -85,B 0,C 180,E1 -2608.577,E2 -2608.577} C_VEL
LIN {X 0,Y 565.836,Z 557.5,A -85,B 0,C 180,E1 -2610,E2 -2610} C_VEL
LIN {X 0,Y 565.843,Z 556.91,A -85,B 0,C 180,E1 -2611.424,E2 -2611.424} C_VEL
LIN {X 0,Y 565.873,Z 555.185,A -85,B 0,C 180,E1 -2612.848,E2 -2612.848} C_VEL
LIN {X 0,Y 565.912,Z 552.289,A -85,B 0,C 180,E1 -2614.273,E2 -2614.273} C_VEL
LIN {X 0,Y 565.982,Z 548.163,A -85,B 0,C 180,E1 -2615.701,E2 -2615.701} C_VEL
LIN {X 0,Y 565.974,Z 542.701,A -85,B 0,C 180,E1 -2617.133,E2 -2617.133} C_VEL
LIN {X 0,Y 566.061,Z 535.747,A -85,B 0,C 180,E1 -2618.568,E2 -2618.568} C_VEL
LIN {X 0,Y 566.177,Z 527.086,A -85,B 0,C 180,E1 -2620.008,E2 -2620.008} C_VEL
LIN {X 0,Y 566.264,Z 518.539,A -85,B 0,C 180,E1 -2621.191,E2 -2621.191} C_VEL
LIN {X 0,Y 566.447,Z 508.506,A -85,B 0,C 180,E1 -2622.358,E2 -2622.358} C_VEL
LIN {X 0,Y 566.65,Z 497.383,A -85,B 0,C 180,E1 -2623.448,E2 -2623.448} C_VEL
LIN {X 0,Y 566.893,Z 484.585,A -85,B 0,C 180,E1 -2624.494,E2 -2624.494} C_VEL
LIN {X 0,Y 567.133,Z 471.773,A -85,B 0,C 180,E1 -2625.36,E2 -2625.36} C_VEL
LIN {X 0,Y 567.387,Z 458.594,A -85,B 0,C 180,E1 -2626.09,E2 -2626.09} C_VEL
LIN {X 0,Y 567.601,Z 444.172,A -85,B 0,C 180,E1 -2626.731,E2 -2626.731} C_VEL
LIN {X 0,Y 567.806,Z 429.245,A -85,B 0,C 180,E1 -2627.235,E2 -2627.235} C_VEL
LIN {X 0,Y 567.911,Z 414.289,A -85,B 0,C 180,E1 -2627.592,E2 -2627.592} C_VEL
LIN {X 0,Y 567.843,Z 402.932,A -85,B 0,C 180,E1 -2627.776,E2 -2627.776} C_VEL
LIN {X 0,Y 566.677,Z 396.801,A -85,B 0,C 180,E1 -2627.897,E2 -2627.897} C_VEL
LIN {X 0,Y 566.921,Z 377.749,A -85,B 0,C 180,E1 -2630.69,E2 -2630.69} C_VEL
LIN {X 0,Y 567.227,Z 358.717,A -85,B 0,C 180,E1 -2633.528,E2 -2633.528} C_VEL
LIN {X 0,Y 567.56,Z 339.363,A -85,B 0,C 180,E1 -2636.474,E2 -2636.474} C_VEL
LIN {X 0,Y 567.75,Z 323.367,A -85,B 0,C 180,E1 -2638.867,E2 -2638.867} C_VEL
LIN {X 0,Y 567.88,Z 315.089,A -85,B 0,C 180,E1 -2640.165,E2 -2640.165} C_VEL
LIN {X 0,Y 568.487,Z 299.752,A -85,B 0,C 180,E1 -2642.79,E2 -2642.79} C_VEL
LIN {X 0,Y 569.032,Z 291.668,A -85,B 0,C 180,E1 -2644.313,E2 -2644.313} C_VEL
LIN {X 0,Y 567.352,Z 284.921,A -85,B 0,C 180,E1 -2645.948,E2 -2645.948} C_VEL
LIN {X 0,Y 566.219,Z 280.583,A -85,B 0,C 180,E1 -2647.205,E2 -2647.205} C_VEL
LIN {X 0,Y 566.211,Z 280.584,A -85,B 0,C 180,E1 -2650.199,E2 -2650.199} C_VEL
LIN {X 0,Y 566.206,Z 280.583,A -85,B 0,C 180,E1 -2653.054,E2 -2653.054} C_VEL
LIN {X 0,Y 566.196,Z 280.584,A -85,B 0,C 180,E1 -2656.049,E2 -2656.049} C_VEL
LIN {X 0,Y 566.177,Z 280.587,A -85,B 0,C 180,E1 -2658.861,E2 -2658.861} C_VEL
LIN {X 0,Y 566.189,Z 280.586,A -85,B 0,C 180,E1 -2661.637,E2 -2661.637} C_VEL
LIN {X 0,Y 566.169,Z 280.59,A -85,B 0,C 180,E1 -2663.791,E2 -2663.791} C_VEL
LIN {X 0,Y 566.23,Z 282.035,A -85,B 0,C 180,E1 -2665.184,E2 -2665.184} C_VEL
LIN {X 0,Y 566.242,Z 284.887,A -85,B 0,C 180,E1 -2667.744,E2 -2667.744} C_VEL
LIN {X 0,Y 566.236,Z 287.51,A -85,B 0,C 180,E1 -2670.323,E2 -2670.323} C_VEL
LIN {X 0,Y 566.2,Z 289.691,A -85,B 0,C 180,E1 -2672.66,E2 -2672.66} C_VEL
LIN {X 0,Y 566.124,Z 291.75,A -85,B 0,C 180,E1 -2675.034,E2 -2675.034} C_VEL
LIN {X 0,Y 566.002,Z 293.656,A -85,B 0,C 180,E1 -2677.361,E2 -2677.361} C_VEL
LIN {X 0,Y 565.969,Z 295.665,A -85,B 0,C 180,E1 -2679.654,E2 -2679.654} C_VEL
LIN {X 0,Y 565.865,Z 297.603,A -85,B 0,C 180,E1 -2681.911,E2 -2681.911} C_VEL
LIN {X 0,Y 565.856,Z 300.306,A -85,B 0,C 180,E1 -2684.143,E2 -2684.143} C_VEL
LIN {X 0,Y 565.883,Z 303.01,A -85,B 0,C 180,E1 -2686.351,E2 -2686.351} C_VEL
LIN {X 0,Y 565.873,Z 304.334,A -85,B 0,C 180,E1 -2687.424,E2 -2687.424} C_VEL
LIN {X 0,Y 566.904,Z 311.794,A -85,B 0,C 180,E1 -2687.629,E2 -2687.629} C_VEL
LIN {X 0,Y 566.753,Z 324.291,A -85,B 0,C 180,E1 -2688.012,E2 -2688.012} C_VEL
LIN {X 0,Y 566.661,Z 336.796,A -85,B 0,C 180,E1 -2688.554,E2 -2688.554} C_VEL
LIN {X 0,Y 566.551,Z 348.083,A -85,B 0,C 180,E1 -2689.193,E2 -2689.193} C_VEL
LIN {X 0,Y 566.345,Z 359.345,A -85,B 0,C 180,E1 -2689.995,E2 -2689.995} C_VEL
LIN {X 0,Y 566.238,Z 369.39,A -85,B 0,C 180,E1 -2690.895,E2 -2690.895} C_VEL
LIN {X 0,Y 566.113,Z 379.092,A -85,B 0,C 180,E1 -2691.972,E2 -2691.972} C_VEL
LIN {X 0,Y 566.05,Z 385.657,A -85,B 0,C 180,E1 -2692.868,E2 -2692.868} C_VEL
LIN {X 0,Y 566.003,Z 392.126,A -85,B 0,C 180,E1 -2693.942,E2 -2693.942} C_VEL
LIN {X 0,Y 565.877,Z 397.265,A -85,B 0,C 180,E1 -2695.013,E2 -2695.013} C_VEL
LIN {X 0,Y 565.927,Z 401.254,A -85,B 0,C 180,E1 -2696.084,E2 -2696.084} C_VEL
LIN {X 0,Y 565.878,Z 404.201,A -85,B 0,C 180,E1 -2697.153,E2 -2697.153} C_VEL
LIN {X 0,Y 565.839,Z 405.627,A -85,B 0,C 180,E1 -2697.865,E2 -2697.865} C_VEL
LIN {X 0,Y 565.842,Z 407.256,A -85,B 0,C 180,E1 -2699.288,E2 -2699.288} C_VEL
LIN {X 0,Y 565.839,Z 407.496,A -85,B 0,C 180,E1 -2700,E2 -2700} C_VEL
LIN {X 0,Y 565.841,Z 407.315,A -85,B 0,C 180,E1 -2700.712,E2 -2700.712} C_VEL
LIN {X 0,Y 565.838,Z 405.77,A -85,B 0,C 180,E1 -2702.136,E2 -2702.136} C_VEL
LIN {X 0,Y 565.879,Z 404.41,A -85,B 0,C 180,E1 -2702.848,E2 -2702.848} C_VEL
LIN {X 0,Y 565.926,Z 401.53,A -85,B 0,C 180,E1 -2703.917,E2 -2703.917} C_VEL
LIN {X 0,Y 565.878,Z 397.628,A -85,B 0,C 180,E1 -2704.988,E2 -2704.988} C_VEL
LIN {X 0,Y 565.99,Z 392.598,A -85,B 0,C 180,E1 -2706.059,E2 -2706.059} C_VEL
LIN {X 0,Y 566.031,Z 386.271,A -85,B 0,C 180,E1 -2707.132,E2 -2707.132} C_VEL
LIN {X 0,Y 566.128,Z 378.349,A -85,B 0,C 180,E1 -2708.208,E2 -2708.208} C_VEL
LIN {X 0,Y 566.249,Z 368.497,A -85,B 0,C 180,E1 -2709.285,E2 -2709.285} C_VEL
LIN {X 0,Y 566.417,Z 358.174,A -85,B 0,C 180,E1 -2710.184,E2 -2710.184} C_VEL
LIN {X 0,Y 566.56,Z 346.895,A -85,B 0,C 180,E1 -2710.972,E2 -2710.972} C_VEL
LIN {X 0,Y 566.687,Z 335.686,A -85,B 0,C 180,E1 -2711.592,E2 -2711.592} C_VEL
LIN {X 0,Y 566.775,Z 324.51,A -85,B 0,C 180,E1 -2712.069,E2 -2712.069} C_VEL
LIN {X 0,Y 566.896,Z 311.741,A -85,B 0,C 180,E1 -2712.462,E2 -2712.462} C_VEL
LIN {X 0,Y 565.878,Z 304.332,A -85,B 0,C 180,E1 -2712.667,E2 -2712.667} C_VEL
LIN {X 0,Y 565.854,Z 301.317,A -85,B 0,C 180,E1 -2715.119,E2 -2715.119} C_VEL
LIN {X 0,Y 565.864,Z 297.711,A -85,B 0,C 180,E1 -2718.089,E2 -2718.089} C_VEL
LIN {X 0,Y 565.905,Z 295.159,A -85,B 0,C 180,E1 -2720.467,E2 -2720.467} C_VEL
LIN {X 0,Y 565.923,Z 291.817,A -85,B 0,C 180,E1 -2723.547,E2 -2723.547} C_VEL
LIN {X 0,Y 565.243,Z 291.272,A -85,B 0,C 180,E1 -2724.138,E2 -2724.138} C_VEL
LIN {X 0,Y 562.374,Z 290.549,A -85,B 0,C 180,E1 -2725.1,E2 -2725.1} C_VEL
LIN {X 0,Y 559.974,Z 289.975,A -85,B 0,C 180,E1 -2725.874,E2 -2725.874} C_VEL
LIN {X 0,Y 558.971,Z 289.422,A -85,B 0,C 180,E1 -2726.471,E2 -2726.471} C_VEL
LIN {X 0,Y 558.904,Z 289.204,A -85,B 0,C 180,E1 -2726.672,E2 -2726.672} C_VEL
LIN {X 0,Y 558.938,Z 286.393,A -85,B 0,C 180,E1 -2729.366,E2 -2729.366} C_VEL
LIN {X 0,Y 558.907,Z 283.558,A -85,B 0,C 180,E1 -2731.879,E2 -2731.879} C_VEL
LIN {X 0,Y 558.962,Z 281.487,A -85,B 0,C 180,E1 -2733.917,E2 -2733.917} C_VEL
LIN {X 0,Y 559.137,Z 281.458,A -85,B 0,C 180,E1 -2736.443,E2 -2736.443} C_VEL
LIN {X 0,Y 559.182,Z 281.46,A -85,B 0,C 180,E1 -2738.934,E2 -2738.934} C_VEL
LIN {X 0,Y 559.166,Z 281.453,A -85,B 0,C 180,E1 -2741.77,E2 -2741.77} C_VEL
LIN {X 0,Y 559.134,Z 281.461,A -85,B 0,C 180,E1 -2744.74,E2 -2744.74} C_VEL
LIN {X 0,Y 559.146,Z 281.464,A -85,B 0,C 180,E1 -2747.866,E2 -2747.866} C_VEL
LIN {X 0,Y 559.094,Z 281.466,A -85,B 0,C 180,E1 -2749.182,E2 -2749.182} C_VEL
LIN {X 0,Y 559.115,Z 282.164,A -85,B 0,C 180,E1 -2750.129,E2 -2750.129} C_VEL
LIN {X 0,Y 559.095,Z 286.665,A -85,B 0,C 180,E1 -2752.888,E2 -2752.888} C_VEL
LIN {X 0,Y 559.045,Z 290.566,A -85,B 0,C 180,E1 -2755.548,E2 -2755.548} C_VEL
LIN {X 0,Y 559.041,Z 295.045,A -85,B 0,C 180,E1 -2758.745,E2 -2758.745} C_VEL
LIN {X 0,Y 558.981,Z 299.212,A -85,B 0,C 180,E1 -2761.655,E2 -2761.655} C_VEL
LIN {X 0,Y 558.925,Z 302.404,A -85,B 0,C 180,E1 -2763.89,E2 -2763.89} C_VEL
LIN {X 0,Y 558.878,Z 306.203,A -85,B 0,C 180,E1 -2766.634,E2 -2766.634} C_VEL
LIN {X 0,Y 558.809,Z 310.346,A -85,B 0,C 180,E1 -2769.381,E2 -2769.381} C_VEL
LIN {X 0,Y 558.815,Z 314.385,A -85,B 0,C 180,E1 -2771.93,E2 -2771.93} C_VEL
LIN {X 0,Y 558.808,Z 314.522,A -85,B 0,C 180,E1 -2771.993,E2 -2771.993} C_VEL
LIN {X 0,Y 561.204,Z 324.702,A -85,B 0,C 180,E1 -2772.242,E2 -2772.242} C_VEL
LIN {X 0,Y 561.006,Z 340.788,A -85,B 0,C 180,E1 -2772.643,E2 -2772.643} C_VEL
LIN {X 0,Y 560.756,Z 353.671,A -85,B 0,C 180,E1 -2773.088,E2 -2773.088} C_VEL
LIN {X 0,Y 560.58,Z 365.718,A -85,B 0,C 180,E1 -2773.615,E2 -2773.615} C_VEL
LIN {X 0,Y 560.346,Z 377.857,A -85,B 0,C 180,E1 -2774.263,E2 -2774.263} C_VEL
LIN {X 0,Y 560.057,Z 390.507,A -85,B 0,C 180,E1 -2775.073,E2 -2775.073} C_VEL
LIN {X 0,Y 559.8,Z 403.72,A -85,B 0,C 180,E1 -2776.107,E2 -2776.107} C_VEL
LIN {X 0,Y 559.558,Z 414.487,A -85,B 0,C 180,E1 -2777.118,E2 -2777.118} C_VEL
LIN {X 0,Y 559.313,Z 424.494,A -85,B 0,C 180,E1 -2778.218,E2 -2778.218} C_VEL
LIN {X 0,Y 559.179,Z 434.334,A -85,B 0,C 180,E1 -2779.499,E2 -2779.499} C_VEL
LIN {X 0,Y 559.003,Z 443.462,A -85,B 0,C 180,E1 -2780.958,E2 -2780.958} C_VEL
LIN {X 0,Y 558.952,Z 449.183,A -85,B 0,C 180,E1 -2782.05,E2 -2782.05} C_VEL
LIN {X 0,Y 558.847,Z 455.25,A -85,B 0,C 180,E1 -2783.462,E2 -2783.462} C_VEL
LIN {X 0,Y 558.856,Z 459.155,A -85,B 0,C 180,E1 -2784.588,E2 -2784.588} C_VEL
LIN {X 0,Y 558.808,Z 462.16,A -85,B 0,C 180,E1 -2785.672,E2 -2785.672} C_VEL
LIN {X 0,Y 558.793,Z 465.104,A -85,B 0,C 180,E1 -2787.116,E2 -2787.116} C_VEL
LIN {X 0,Y 558.742,Z 466.875,A -85,B 0,C 180,E1 -2788.558,E2 -2788.558} C_VEL
LIN {X 0,Y 558.738,Z 467.496,A -85,B 0,C 180,E1 -2790,E2 -2790} C_VEL
LIN {X 0,Y 558.744,Z 466.96,A -85,B 0,C 180,E1 -2791.441,E2 -2791.441} C_VEL
LIN {X 0,Y 558.795,Z 465.257,A -85,B 0,C 180,E1 -2792.884,E2 -2792.884} C_VEL
LIN {X 0,Y 558.808,Z 462.376,A -85,B 0,C 180,E1 -2794.328,E2 -2794.328} C_VEL
LIN {X 0,Y 558.887,Z 458.309,A -85,B 0,C 180,E1 -2795.774,E2 -2795.774} C_VEL
LIN {X 0,Y 558.899,Z 452.912,A -85,B 0,C 180,E1 -2797.224,E2 -2797.224} C_VEL
LIN {X 0,Y 559,Z 445.959,A -85,B 0,C 180,E1 -2798.677,E2 -2798.677} C_VEL
LIN {X 0,Y 559.091,Z 438.523,A -85,B 0,C 180,E1 -2799.953,E2 -2799.953} C_VEL
LIN {X 0,Y 559.2,Z 430.892,A -85,B 0,C 180,E1 -2801.059,E2 -2801.059} C_VEL
LIN {X 0,Y 559.381,Z 422.147,A -85,B 0,C 180,E1 -2802.148,E2 -2802.148} C_VEL
LIN {X 0,Y 559.619,Z 411.776,A -85,B 0,C 180,E1 -2803.249,E2 -2803.249} C_VEL
LIN {X 0,Y 559.859,Z 399.24,A -85,B 0,C 180,E1 -2804.355,E2 -2804.355} C_VEL
LIN {X 0,Y 560.164,Z 387.75,A -85,B 0,C 180,E1 -2805.202,E2 -2805.202} C_VEL
LIN {X 0,Y 560.364,Z 376.202,A -85,B 0,C 180,E1 -2805.923,E2 -2805.923} C_VEL
LIN {X 0,Y 560.615,Z 363.748,A -85,B 0,C 180,E1 -2806.571,E2 -2806.571} C_VEL
LIN {X 0,Y 560.91,Z 348.905,A -85,B 0,C 180,E1 -2807.184,E2 -2807.184} C_VEL
LIN {X 0,Y 561.085,Z 333.748,A -85,B 0,C 180,E1 -2807.641,E2 -2807.641} C_VEL
LIN {X 0,Y 561.067,Z 323.922,A -85,B 0,C 180,E1 -2807.866,E2 -2807.866} C_VEL
LIN {X 0,Y 558.827,Z 314.482,A -85,B 0,C 180,E1 -2808.099,E2 -2808.099} C_VEL
LIN {X 0,Y 558.808,Z 310.488,A -85,B 0,C 180,E1 -2810.619,E2 -2810.619} C_VEL
LIN {X 0,Y 558.876,Z 306.337,A -85,B 0,C 180,E1 -2813.365,E2 -2813.365} C_VEL
LIN {X 0,Y 558.925,Z 302.519,A -85,B 0,C 180,E1 -2816.11,E2 -2816.11} C_VEL
LIN {X 0,Y 559.014,Z 299.07,A -85,B 0,C 180,E1 -2818.538,E2 -2818.538} C_VEL
LIN {X 0,Y 559.042,Z 295.174,A -85,B 0,C 180,E1 -2821.255,E2 -2821.255} C_VEL
LIN {X 0,Y 559.056,Z 290.702,A -85,B 0,C 180,E1 -2824.451,E2 -2824.451} C_VEL
LIN {X 0,Y 559.094,Z 286.803,A -85,B 0,C 180,E1 -2827.112,E2 -2827.112} C_VEL
LIN {X 0,Y 559.095,Z 282.236,A -85,B 0,C 180,E1 -2829.933,E2 -2829.933} C_VEL
LIN {X 0,Y 559.078,Z 281.475,A -85,B 0,C 180,E1 -2830.464,E2 -2830.464} C_VEL
LIN {X 0,Y 559.146,Z 281.461,A -85,B 0,C 180,E1 -2833.196,E2 -2833.196} C_VEL
LIN {X 0,Y 559.139,Z 281.46,A -85,B 0,C 180,E1 -2836.266,E2 -2836.266} C_VEL
LIN {X 0,Y 559.156,Z 281.458,A -85,B 0,C 180,E1 -2839.187,E2 -2839.187} C_VEL
LIN {X 0,Y 559.124,Z 281.468,A -85,B 0,C 180,E1 -2841.982,E2 -2841.982} C_VEL
LIN {X 0,Y 559.146,Z 281.459,A -85,B 0,C 180,E1 -2844.785,E2 -2844.785} C_VEL
LIN {X 0,Y 559.156,Z 281.459,A -85,B 0,C 180,E1 -2847.364,E2 -2847.364} C_VEL
LIN {X 0,Y 559.119,Z 281.465,A -85,B 0,C 180,E1 -2850.148,E2 -2850.148} C_VEL
LIN {X 0,Y 559.116,Z 281.463,A -85,B 0,C 180,E1 -2853.184,E2 -2853.184} C_VEL
LIN {X 0,Y 559.157,Z 281.461,A -85,B 0,C 180,E1 -2855.495,E2 -2855.495} C_VEL
LIN {X 0,Y 559.173,Z 281.458,A -85,B 0,C 180,E1 -2858.624,E2 -2858.624} C_VEL
LIN {X 0,Y 559.157,Z 281.457,A -85,B 0,C 180,E1 -2860.926,E2 -2860.926} C_VEL
LIN {X 0,Y 559.141,Z 281.46,A -85,B 0,C 180,E1 -2863.947,E2 -2863.947} C_VEL
LIN {X 0,Y 559.173,Z 281.455,A -85,B 0,C 180,E1 -2866.184,E2 -2866.184} C_VEL
LIN {X 0,Y 559.196,Z 281.451,A -85,B 0,C 180,E1 -2869.133,E2 -2869.133} C_VEL
LIN {X 0,Y 559.171,Z 281.459,A -85,B 0,C 180,E1 -2872.053,E2 -2872.053} C_VEL
LIN {X 0,Y 559.243,Z 281.446,A -85,B 0,C 180,E1 -2874.953,E2 -2874.953} C_VEL
LIN {X 0,Y 559.248,Z 281.445,A -85,B 0,C 180,E1 -2877.839,E2 -2877.839} C_VEL
LIN {X 0,Y 559.269,Z 281.443,A -85,B 0,C 180,E1 -2880.72,E2 -2880.72} C_VEL
LIN {X 0,Y 559.223,Z 281.448,A -85,B 0,C 180,E1 -2882.881,E2 -2882.881} C_VEL
LIN {X 0,Y 559.213,Z 281.448,A -85,B 0,C 180,E1 -2885.77,E2 -2885.77} C_VEL
LIN {X 0,Y 559.173,Z 281.46,A -85,B 0,C 180,E1 -2888.675,E2 -2888.675} C_VEL
LIN {X 0,Y 559.206,Z 281.449,A -85,B 0,C 180,E1 -2891.6,E2 -2891.6} C_VEL
LIN {X 0,Y 559.152,Z 281.457,A -85,B 0,C 180,E1 -2894.576,E2 -2894.576} C_VEL
LIN {X 0,Y 559.135,Z 281.459,A -85,B 0,C 180,E1 -2897.558,E2 -2897.558} C_VEL
LIN {X 0,Y 559.173,Z 281.457,A -85,B 0,C 180,E1 -2899.837,E2 -2899.837} C_VEL
LIN {X 0,Y 559.14,Z 281.461,A -85,B 0,C 180,E1 -2902.153,E2 -2902.153} C_VEL
LIN {X 0,Y 559.138,Z 281.465,A -85,B 0,C 180,E1 -2905.178,E2 -2905.178} C_VEL
LIN {X 0,Y 559.127,Z 281.459,A -85,B 0,C 180,E1 -2907.715,E2 -2907.715} C_VEL
LIN {X 0,Y 559.155,Z 281.463,A -85,B 0,C 180,E1 -2910.183,E2 -2910.183} C_VEL
LIN {X 0,Y 559.157,Z 281.456,A -85,B 0,C 180,E1 -2912.715,E2 -2912.715} C_VEL
LIN {X 0,Y 559.122,Z 281.467,A -85,B 0,C 180,E1 -2915.324,E2 -2915.324} C_VEL
LIN {X 0,Y 559.123,Z 281.462,A -85,B 0,C 180,E1 -2918.018,E2 -2918.018} C_VEL
LIN {X 0,Y 559.156,Z 281.457,A -85,B 0,C 180,E1 -2920.812,E2 -2920.812} C_VEL
LIN {X 0,Y 559.145,Z 281.46,A -85,B 0,C 180,E1 -2923.196,E2 -2923.196} C_VEL
LIN {X 0,Y 559.134,Z 281.459,A -85,B 0,C 180,E1 -2926.266,E2 -2926.266} C_VEL
LIN {X 0,Y 559.151,Z 281.459,A -85,B 0,C 180,E1 -2929.187,E2 -2929.187} C_VEL
LIN {X 0,Y 559.133,Z 281.469,A -85,B 0,C 180,E1 -2931.983,E2 -2931.983} C_VEL
LIN {X 0,Y 559.161,Z 281.533,A -85,B 0,C 180,E1 -2933.394,E2 -2933.394} C_VEL
LIN {X 0,Y 561.564,Z 290.975,A -85,B 0,C 180,E1 -2935.29,E2 -2935.29} C_VEL
LIN {X 0,Y 561.888,Z 294.668,A -85,B 0,C 180,E1 -2935.963,E2 -2935.963} C_VEL
LIN {X 0,Y 561.285,Z 312.061,A -85,B 0,C 180,E1 -2938.911,E2 -2938.911} C_VEL
LIN {X 0,Y 560.895,Z 331.385,A -85,B 0,C 180,E1 -2941.974,E2 -2941.974} C_VEL
LIN {X 0,Y 560.537,Z 349.58,A -85,B 0,C 180,E1 -2944.768,E2 -2944.768} C_VEL
LIN {X 0,Y 560.181,Z 368.795,A -85,B 0,C 180,E1 -2947.696,E2 -2947.696} C_VEL
LIN {X 0,Y 559.861,Z 388.397,A -85,B 0,C 180,E1 -2950.631,E2 -2950.631} C_VEL
LIN {X 0,Y 559.74,Z 396.748,A -85,B 0,C 180,E1 -2951.866,E2 -2951.866} C_VEL
LIN {X 0,Y 561.223,Z 404.734,A -85,B 0,C 180,E1 -2952.031,E2 -2952.031} C_VEL
LIN {X 0,Y 561.099,Z 420.691,A -85,B 0,C 180,E1 -2952.324,E2 -2952.324} C_VEL
LIN {X 0,Y 560.96,Z 435.295,A -85,B 0,C 180,E1 -2952.736,E2 -2952.736} C_VEL
LIN {X 0,Y 560.716,Z 449.801,A -85,B 0,C 180,E1 -2953.292,E2 -2953.292} C_VEL
LIN {X 0,Y 560.433,Z 463.879,A -85,B 0,C 180,E1 -2953.985,E2 -2953.985} C_VEL
LIN {X 0,Y 560.183,Z 476.047,A -85,B 0,C 180,E1 -2954.724,E2 -2954.724} C_VEL
LIN {X 0,Y 559.881,Z 488.701,A -85,B 0,C 180,E1 -2955.646,E2 -2955.646} C_VEL
LIN {X 0,Y 559.659,Z 499.333,A -85,B 0,C 180,E1 -2956.567,E2 -2956.567} C_VEL
LIN {X 0,Y 559.412,Z 510.141,A -85,B 0,C 180,E1 -2957.668,E2 -2957.668} C_VEL
LIN {X 0,Y 559.239,Z 520.635,A -85,B 0,C 180,E1 -2958.947,E2 -2958.947} C_VEL
LIN {X 0,Y 559.077,Z 529.418,A -85,B 0,C 180,E1 -2960.229,E2 -2960.229} C_VEL
LIN {X 0,Y 559,Z 535.75,A -85,B 0,C 180,E1 -2961.323,E2 -2961.323} C_VEL
LIN {X 0,Y 558.899,Z 542.701,A -85,B 0,C 180,E1 -2962.776,E2 -2962.776} C_VEL
LIN {X 0,Y 558.888,Z 548.161,A -85,B 0,C 180,E1 -2964.226,E2 -2964.226} C_VEL
LIN {X 0,Y 558.807,Z 552.291,A -85,B 0,C 180,E1 -2965.672,E2 -2965.672} C_VEL
LIN {X 0,Y 558.794,Z 555.187,A -85,B 0,C 180,E1 -2967.116,E2 -2967.116} C_VEL
LIN {X 0,Y 558.743,Z 556.911,A -85,B 0,C 180,E1 -2968.559,E2 -2968.559} C_VEL
LIN {X 0,Y 558.737,Z 557.5,A -85,B 0,C 180,E1 -2970,E2 -2970} C_VEL
LIN {X 0,Y 558.743,Z 556.91,A -85,B 0,C 180,E1 -2971.442,E2 -2971.442} C_VEL
LIN {X 0,Y 558.794,Z 555.184,A -85,B 0,C 180,E1 -2972.884,E2 -2972.884} C_VEL
LIN {X 0,Y 558.807,Z 552.289,A -85,B 0,C 180,E1 -2974.328,E2 -2974.328} C_VEL
LIN {X 0,Y 558.888,Z 548.163,A -85,B 0,C 180,E1 -2975.774,E2 -2975.774} C_VEL
LIN {X 0,Y 558.9,Z 542.701,A -85,B 0,C 180,E1 -2977.224,E2 -2977.224} C_VEL
LIN {X 0,Y 559.001,Z 535.746,A -85,B 0,C 180,E1 -2978.677,E2 -2978.677} C_VEL
LIN {X 0,Y 559.092,Z 528.291,A -85,B 0,C 180,E1 -2979.953,E2 -2979.953} C_VEL
LIN {X 0,Y 559.228,Z 519.12,A -85,B 0,C 180,E1 -2981.258,E2 -2981.258} C_VEL
LIN {X 0,Y 559.474,Z 508.506,A -85,B 0,C 180,E1 -2982.515,E2 -2982.515} C_VEL
LIN {X 0,Y 559.693,Z 496.352,A -85,B 0,C 180,E1 -2983.71,E2 -2983.71} C_VEL
LIN {X 0,Y 560.003,Z 483.521,A -85,B 0,C 180,E1 -2984.754,E2 -2984.754} C_VEL
LIN {X 0,Y 560.303,Z 470.241,A -85,B 0,C 180,E1 -2985.645,E2 -2985.645} C_VEL
LIN {X 0,Y 560.567,Z 456.763,A -85,B 0,C 180,E1 -2986.385,E2 -2986.385} C_VEL
LIN {X 0,Y 560.834,Z 443.04,A -85,B 0,C 180,E1 -2986.986,E2 -2986.986} C_VEL
LIN {X 0,Y 561.033,Z 427.709,A -85,B 0,C 180,E1 -2987.497,E2 -2987.497} C_VEL
LIN {X 0,Y 561.225,Z 412.149,A -85,B 0,C 180,E1 -2987.852,E2 -2987.852} C_VEL
LIN {X 0,Y 561.091,Z 403.841,A -85,B 0,C 180,E1 -2987.985,E2 -2987.985} C_VEL
LIN {X 0,Y 559.741,Z 396.744,A -85,B 0,C 180,E1 -2988.134,E2 -2988.134} C_VEL
LIN {X 0,Y 560.056,Z 376.47,A -85,B 0,C 180,E1 -2991.148,E2 -2991.148} C_VEL
LIN {X 0,Y 560.385,Z 357.279,A -85,B 0,C 180,E1 -2994.054,E2 -2994.054} C_VEL
LIN {X 0,Y 560.638,Z 340.247,A -85,B 0,C 180,E1 -2996.625,E2 -2996.625} C_VEL
LIN {X 0,Y 560.868,Z 323.971,A -85,B 0,C 180,E1 -2999.087,E2 -2999.087} C_VEL
LIN {X 0,Y 561.436,Z 307.047,A -85,B 0,C 180,E1 -3001.93,E2 -3001.93} C_VEL
LIN {X 0,Y 562.299,Z 294.77,A -85,B 0,C 180,E1 -3004.225,E2 -3004.225} C_VEL
LIN {X 0,Y 562.083,Z 292.602,A -85,B 0,C 180,E1 -3004.702,E2 -3004.702} C_VEL
LIN {X 0,Y 560.641,Z 287.115,A -85,B 0,C 180,E1 -3006.099,E2 -3006.099} C_VEL
LIN {X 0,Y 559.128,Z 281.465,A -85,B 0,C 180,E1 -3007.854,E2 -3007.854} C_VEL
LIN {X 0,Y 559.166,Z 281.461,A -85,B 0,C 180,E1 -3009.942,E2 -3009.942} C_VEL
LIN {X 0,Y 559.161,Z 281.462,A -85,B 0,C 180,E1 -3012.744,E2 -3012.744} C_VEL
LIN {X 0,Y 559.149,Z 281.462,A -85,B 0,C 180,E1 -3015.762,E2 -3015.762} C_VEL
LIN {X 0,Y 559.168,Z 281.461,A -85,B 0,C 180,E1 -3018.23,E2 -3018.23} C_VEL
LIN {X 0,Y 559.177,Z 281.459,A -85,B 0,C 180,E1 -3021.192,E2 -3021.192} C_VEL
LIN {X 0,Y 559.133,Z 281.543,A -85,B 0,C 180,E1 -3023.789,E2 -3023.789} C_VEL
LIN {X 0,Y 559.263,Z 284.612,A -85,B 0,C 180,E1 -3026.432,E2 -3026.432} C_VEL
LIN {X 0,Y 559.199,Z 287.278,A -85,B 0,C 180,E1 -3028.983,E2 -3028.983} C_VEL
LIN {X 0,Y 559.208,Z 289.784,A -85,B 0,C 180,E1 -3031.612,E2 -3031.612} C_VEL
LIN {X 0,Y 559.14,Z 291.828,A -85,B 0,C 180,E1 -3033.901,E2 -3033.901} C_VEL
LIN {X 0,Y 559.068,Z 294.131,A -85,B 0,C 180,E1 -3036.589,E2 -3036.589} C_VEL
LIN {X 0,Y 558.968,Z 296.523,A -85,B 0,C 180,E1 -3039.387,E2 -3039.387} C_VEL
LIN {X 0,Y 558.845,Z 298.463,A -85,B 0,C 180,E1 -3041.676,E2 -3041.676} C_VEL
LIN {X 0,Y 558.77,Z 300.335,A -85,B 0,C 180,E1 -3043.936,E2 -3043.936} C_VEL
LIN {X 0,Y 558.781,Z 303.011,A -85,B 0,C 180,E1 -3046.174,E2 -3046.174} C_VEL
LIN {X 0,Y 558.784,Z 304.334,A -85,B 0,C 180,E1 -3047.262,E2 -3047.262} C_VEL
LIN {X 0,Y 559.972,Z 312.733,A -85,B 0,C 180,E1 -3047.497,E2 -3047.497} C_VEL
LIN {X 0,Y 559.821,Z 324.809,A -85,B 0,C 180,E1 -3047.88,E2 -3047.88} C_VEL
LIN {X 0,Y 559.688,Z 336.805,A -85,B 0,C 180,E1 -3048.41,E2 -3048.41} C_VEL
LIN {X 0,Y 559.559,Z 348.164,A -85,B 0,C 180,E1 -3049.061,E2 -3049.061} C_VEL
LIN {X 0,Y 559.361,Z 359.354,A -85,B 0,C 180,E1 -3049.869,E2 -3049.869} C_VEL
LIN {X 0,Y 559.211,Z 369.395,A -85,B 0,C 180,E1 -3050.779,E2 -3050.779} C_VEL
LIN {X 0,Y 559.05,Z 379.096,A -85,B 0,C 180,E1 -3051.87,E2 -3051.87} C_VEL
LIN {X 0,Y 558.971,Z 386.954,A -85,B 0,C 180,E1 -3052.977,E2 -3052.977} C_VEL
LIN {X 0,Y 558.936,Z 393.953,A -85,B 0,C 180,E1 -3054.227,E2 -3054.227} C_VEL
LIN {X 0,Y 558.826,Z 398.696,A -85,B 0,C 180,E1 -3055.311,E2 -3055.311} C_VEL
LIN {X 0,Y 558.837,Z 402.327,A -85,B 0,C 180,E1 -3056.395,E2 -3056.395} C_VEL
LIN {X 0,Y 558.799,Z 404.203,A -85,B 0,C 180,E1 -3057.116,E2 -3057.116} C_VEL
LIN {X 0,Y 558.745,Z 405.626,A -85,B 0,C 180,E1 -3057.838,E2 -3057.838} C_VEL
LIN {X 0,Y 558.742,Z 407.257,A -85,B 0,C 180,E1 -3059.279,E2 -3059.279} C_VEL
LIN {X 0,Y 558.74,Z 407.496,A -85,B 0,C 180,E1 -3060,E2 -3060} C_VEL
LIN {X 0,Y 558.741,Z 407.315,A -85,B 0,C 180,E1 -3060.721,E2 -3060.721} C_VEL
LIN {X 0,Y 558.745,Z 405.769,A -85,B 0,C 180,E1 -3062.163,E2 -3062.163} C_VEL
LIN {X 0,Y 558.8,Z 404.408,A -85,B 0,C 180,E1 -3062.884,E2 -3062.884} C_VEL
LIN {X 0,Y 558.844,Z 401.527,A -85,B 0,C 180,E1 -3063.966,E2 -3063.966} C_VEL
LIN {X 0,Y 558.798,Z 397.626,A -85,B 0,C 180,E1 -3065.051,E2 -3065.051} C_VEL
LIN {X 0,Y 558.91,Z 392.596,A -85,B 0,C 180,E1 -3066.136,E2 -3066.136} C_VEL
LIN {X 0,Y 558.973,Z 386.267,A -85,B 0,C 180,E1 -3067.223,E2 -3067.223} C_VEL
LIN {X 0,Y 559.091,Z 378.344,A -85,B 0,C 180,E1 -3068.312,E2 -3068.312} C_VEL
LIN {X 0,Y 559.224,Z 368.491,A -85,B 0,C 180,E1 -3069.403,E2 -3069.403} C_VEL
LIN {X 0,Y 559.41,Z 358.165,A -85,B 0,C 180,E1 -3070.313,E2 -3070.313} C_VEL
LIN {X 0,Y 559.575,Z 347.201,A -85,B 0,C 180,E1 -3071.09,E2 -3071.09} C_VEL
LIN {X 0,Y 559.709,Z 336.951,A -85,B 0,C 180,E1 -3071.672,E2 -3071.672} C_VEL
LIN {X 0,Y 559.809,Z 325.455,A -85,B 0,C 180,E1 -3072.185,E2 -3072.185} C_VEL
LIN {X 0,Y 559.981,Z 312.631,A -85,B 0,C 180,E1 -3072.595,E2 -3072.595} C_VEL
LIN {X 0,Y 558.768,Z 304.331,A -85,B 0,C 180,E1 -3072.831,E2 -3072.831} C_VEL
LIN {X 0,Y 558.752,Z 301.317,A -85,B 0,C 180,E1 -3075.316,E2 -3075.316} C_VEL
LIN {X 0,Y 558.767,Z 298.831,A -85,B 0,C 180,E1 -3077.57,E2 -3077.57} C_VEL
LIN {X 0,Y 558.838,Z 296.5,A -85,B 0,C 180,E1 -3079.85,E2 -3079.85} C_VEL
LIN {X 0,Y 558.827,Z 293.942,A -85,B 0,C 180,E1 -3082.166,E2 -3082.166} C_VEL
LIN {X 0,Y 558.884,Z 290.812,A -85,B 0,C 180,E1 -3085.122,E2 -3085.122} C_VEL
LIN {X 0,Y 558.904,Z 289.204,A -85,B 0,C 180,E1 -3086.672,E2 -3086.672} C_VEL
LIN {X 0,Y 558.283,Z 288.624,A -85,B 0,C 180,E1 -3087.271,E2 -3087.271} C_VEL
LIN {X 0,Y 555.468,Z 287.887,A -85,B 0,C 180,E1 -3088.245,E2 -3088.245} C_VEL
LIN {X 0,Y 553.053,Z 287.308,A -85,B 0,C 180,E1 -3089.03,E2 -3089.03} C_VEL
LIN {X 0,Y 551.995,Z 286.761,A -85,B 0,C 180,E1 -3089.634,E2 -3089.634} C_VEL
LIN {X 0,Y 551.9,Z 286.53,A -85,B 0,C 180,E1 -3089.838,E2 -3089.838} C_VEL
LIN {X 0,Y 551.855,Z 282.749,A -85,B 0,C 180,E1 -3093.204,E2 -3093.204} C_VEL
LIN {X 0,Y 551.942,Z 282.361,A -85,B 0,C 180,E1 -3094.14,E2 -3094.14} C_VEL
LIN {X 0,Y 552.105,Z 282.336,A -85,B 0,C 180,E1 -3096.747,E2 -3096.747} C_VEL
LIN {X 0,Y 552.137,Z 282.331,A -85,B 0,C 180,E1 -3099.527,E2 -3099.527} C_VEL
LIN {X 0,Y 552.133,Z 282.335,A -85,B 0,C 180,E1 -3102.425,E2 -3102.425} C_VEL
LIN {X 0,Y 552.077,Z 282.338,A -85,B 0,C 180,E1 -3105.56,E2 -3105.56} C_VEL
LIN {X 0,Y 552.11,Z 282.337,A -85,B 0,C 180,E1 -3107.587,E2 -3107.587} C_VEL
LIN {X 0,Y 552.024,Z 282.488,A -85,B 0,C 180,E1 -3109.808,E2 -3109.808} C_VEL
LIN {X 0,Y 552.048,Z 286.619,A -85,B 0,C 180,E1 -3112.332,E2 -3112.332} C_VEL
LIN {X 0,Y 552.014,Z 290.649,A -85,B 0,C 180,E1 -3115.046,E2 -3115.046} C_VEL
LIN {X 0,Y 551.963,Z 294.342,A -85,B 0,C 180,E1 -3117.671,E2 -3117.671} C_VEL
LIN {X 0,Y 551.933,Z 297.926,A -85,B 0,C 180,E1 -3120.224,E2 -3120.224} C_VEL
LIN {X 0,Y 551.917,Z 301.965,A -85,B 0,C 180,E1 -3123.045,E2 -3123.045} C_VEL
LIN {X 0,Y 551.822,Z 306.094,A -85,B 0,C 180,E1 -3125.949,E2 -3125.949} C_VEL
LIN {X 0,Y 551.785,Z 309.397,A -85,B 0,C 180,E1 -3128.402,E2 -3128.402} C_VEL
LIN {X 0,Y 551.795,Z 312.767,A -85,B 0,C 180,E1 -3130.661,E2 -3130.661} C_VEL
LIN {X 0,Y 551.726,Z 314.467,A -85,B 0,C 180,E1 -3131.741,E2 -3131.741} C_VEL
LIN {X 0,Y 554.388,Z 325.396,A -85,B 0,C 180,E1 -3132.029,E2 -3132.029} C_VEL
LIN {X 0,Y 554.22,Z 340.956,A -85,B 0,C 180,E1 -3132.429,E2 -3132.429} C_VEL
LIN {X 0,Y 553.963,Z 353.929,A -85,B 0,C 180,E1 -3132.885,E2 -3132.885} C_VEL
LIN {X 0,Y 553.752,Z 365.713,A -85,B 0,C 180,E1 -3133.407,E2 -3133.407} C_VEL
LIN {X 0,Y 553.477,Z 377.853,A -85,B 0,C 180,E1 -3134.062,E2 -3134.062} C_VEL
LIN {X 0,Y 553.192,Z 389.95,A -85,B 0,C 180,E1 -3134.845,E2 -3134.845} C_VEL
LIN {X 0,Y 552.861,Z 403.725,A -85,B 0,C 180,E1 -3135.929,E2 -3135.929} C_VEL
LIN {X 0,Y 552.562,Z 414.485,A -85,B 0,C 180,E1 -3136.952,E2 -3136.952} C_VEL
LIN {X 0,Y 552.353,Z 422.934,A -85,B 0,C 180,E1 -3137.881,E2 -3137.881} C_VEL
LIN {X 0,Y 552.173,Z 431.644,A -85,B 0,C 180,E1 -3138.993,E2 -3138.993} C_VEL
LIN {X 0,Y 552.019,Z 439.109,A -85,B 0,C 180,E1 -3140.103,E2 -3140.103} C_VEL
LIN {X 0,Y 551.91,Z 447.417,A -85,B 0,C 180,E1 -3141.579,E2 -3141.579} C_VEL
LIN {X 0,Y 551.814,Z 453.993,A -85,B 0,C 180,E1 -3143.05,E2 -3143.05} C_VEL
LIN {X 0,Y 551.786,Z 459.15,A -85,B 0,C 180,E1 -3144.518,E2 -3144.518} C_VEL
LIN {X 0,Y 551.73,Z 463.82,A -85,B 0,C 180,E1 -3146.348,E2 -3146.348} C_VEL
LIN {X 0,Y 551.655,Z 466.133,A -85,B 0,C 180,E1 -3147.809,E2 -3147.809} C_VEL
LIN {X 0,Y 551.637,Z 467.289,A -85,B 0,C 180,E1 -3149.27,E2 -3149.27} C_VEL
LIN {X 0,Y 551.638,Z 467.319,A -85,B 0,C 180,E1 -3150.73,E2 -3150.73} C_VEL
LIN {X 0,Y 551.656,Z 466.229,A -85,B 0,C 180,E1 -3152.19,E2 -3152.19} C_VEL
LIN {X 0,Y 551.731,Z 463.997,A -85,B 0,C 180,E1 -3153.652,E2 -3153.652} C_VEL
LIN {X 0,Y 551.786,Z 459.428,A -85,B 0,C 180,E1 -3155.481,E2 -3155.481} C_VEL
LIN {X 0,Y 551.781,Z 455.741,A -85,B 0,C 180,E1 -3156.582,E2 -3156.582} C_VEL
LIN {X 0,Y 551.831,Z 451.284,A -85,B 0,C 180,E1 -3157.685,E2 -3157.685} C_VEL
LIN {X 0,Y 551.921,Z 444.95,A -85,B 0,C 180,E1 -3158.974,E2 -3158.974} C_VEL
LIN {X 0,Y 552.07,Z 438.511,A -85,B 0,C 180,E1 -3160.081,E2 -3160.081} C_VEL
LIN {X 0,Y 552.154,Z 431.148,A -85,B 0,C 180,E1 -3161.165,E2 -3161.165} C_VEL
LIN {X 0,Y 552.377,Z 422.133,A -85,B 0,C 180,E1 -3162.305,E2 -3162.305} C_VEL
LIN {X 0,Y 552.633,Z 411.769,A -85,B 0,C 180,E1 -3163.42,E2 -3163.42} C_VEL
LIN {X 0,Y 552.929,Z 399.222,A -85,B 0,C 180,E1 -3164.538,E2 -3164.538} C_VEL
LIN {X 0,Y 553.223,Z 388.843,A -85,B 0,C 180,E1 -3165.32,E2 -3165.32} C_VEL
LIN {X 0,Y 553.468,Z 377.781,A -85,B 0,C 180,E1 -3166.032,E2 -3166.032} C_VEL
LIN {X 0,Y 553.727,Z 365.622,A -85,B 0,C 180,E1 -3166.688,E2 -3166.688} C_VEL
LIN {X 0,Y 554.01,Z 353.686,A -85,B 0,C 180,E1 -3167.213,E2 -3167.213} C_VEL
LIN {X 0,Y 554.218,Z 339.932,A -85,B 0,C 180,E1 -3167.695,E2 -3167.695} C_VEL
LIN {X 0,Y 554.28,Z 324.952,A -85,B 0,C 180,E1 -3168.073,E2 -3168.073} C_VEL
LIN {X 0,Y 551.738,Z 314.481,A -85,B 0,C 180,E1 -3168.339,E2 -3168.339} C_VEL
LIN {X 0,Y 551.748,Z 310.498,A -85,B 0,C 180,E1 -3170.895,E2 -3170.895} C_VEL
LIN {X 0,Y 551.829,Z 306.989,A -85,B 0,C 180,E1 -3173.511,E2 -3173.511} C_VEL
LIN {X 0,Y 551.879,Z 302.788,A -85,B 0,C 180,E1 -3176.469,E2 -3176.469} C_VEL
LIN {X 0,Y 551.929,Z 299.258,A -85,B 0,C 180,E1 -3178.939,E2 -3178.939} C_VEL
LIN {X 0,Y 551.998,Z 295.657,A -85,B 0,C 180,E1 -3181.467,E2 -3181.467} C_VEL
LIN {X 0,Y 552.011,Z 291.934,A -85,B 0,C 180,E1 -3184.151,E2 -3184.151} C_VEL
LIN {X 0,Y 552.041,Z 288.174,A -85,B 0,C 180,E1 -3186.752,E2 -3186.752} C_VEL
LIN {X 0,Y 552.054,Z 283.772,A -85,B 0,C 180,E1 -3189.534,E2 -3189.534} C_VEL
LIN {X 0,Y 552.034,Z 282.353,A -85,B 0,C 180,E1 -3190.488,E2 -3190.488} C_VEL
LIN {X 0,Y 552.108,Z 282.34,A -85,B 0,C 180,E1 -3193.424,E2 -3193.424} C_VEL
LIN {X 0,Y 552.107,Z 282.338,A -85,B 0,C 180,E1 -3196.576,E2 -3196.576} C_VEL
LIN {X 0,Y 552.107,Z 282.335,A -85,B 0,C 180,E1 -3199.519,E2 -3199.519} C_VEL
LIN {X 0,Y 552.083,Z 282.34,A -85,B 0,C 180,E1 -3202.335,E2 -3202.335} C_VEL
LIN {X 0,Y 552.119,Z 282.337,A -85,B 0,C 180,E1 -3205.053,E2 -3205.053} C_VEL
LIN {X 0,Y 552.116,Z 282.334,A -85,B 0,C 180,E1 -3207.681,E2 -3207.681} C_VEL
LIN {X 0,Y 552.082,Z 282.342,A -85,B 0,C 180,E1 -3210.233,E2 -3210.233} C_VEL
LIN {X 0,Y 552.077,Z 282.339,A -85,B 0,C 180,E1 -3213.013,E2 -3213.013} C_VEL
LIN {X 0,Y 552.105,Z 282.339,A -85,B 0,C 180,E1 -3215.161,E2 -3215.161} C_VEL
LIN {X 0,Y 552.127,Z 282.334,A -85,B 0,C 180,E1 -3218.337,E2 -3218.337} C_VEL
LIN {X 0,Y 552.149,Z 282.331,A -85,B 0,C 180,E1 -3220.674,E2 -3220.674} C_VEL
LIN {X 0,Y 552.088,Z 282.341,A -85,B 0,C 180,E1 -3223.736,E2 -3223.736} C_VEL
LIN {X 0,Y 552.137,Z 282.331,A -85,B 0,C 180,E1 -3226.004,E2 -3226.004} C_VEL
LIN {X 0,Y 552.164,Z 282.328,A -85,B 0,C 180,E1 -3228.993,E2 -3228.993} C_VEL
LIN {X 0,Y 552.132,Z 282.337,A -85,B 0,C 180,E1 -3231.951,E2 -3231.951} C_VEL
LIN {X 0,Y 552.217,Z 282.32,A -85,B 0,C 180,E1 -3234.889,E2 -3234.889} C_VEL
LIN {X 0,Y 552.22,Z 282.32,A -85,B 0,C 180,E1 -3237.812,E2 -3237.812} C_VEL
LIN {X 0,Y 552.24,Z 282.318,A -85,B 0,C 180,E1 -3240.729,E2 -3240.729} C_VEL
LIN {X 0,Y 552.191,Z 282.325,A -85,B 0,C 180,E1 -3242.918,E2 -3242.918} C_VEL
LIN {X 0,Y 552.182,Z 282.323,A -85,B 0,C 180,E1 -3245.844,E2 -3245.844} C_VEL
LIN {X 0,Y 552.149,Z 282.333,A -85,B 0,C 180,E1 -3248.786,E2 -3248.786} C_VEL
LIN {X 0,Y 552.162,Z 282.328,A -85,B 0,C 180,E1 -3251.75,E2 -3251.75} C_VEL
LIN {X 0,Y 552.119,Z 282.334,A -85,B 0,C 180,E1 -3254.749,E2 -3254.749} C_VEL
LIN {X 0,Y 552.095,Z 282.335,A -85,B 0,C 180,E1 -3257.789,E2 -3257.789} C_VEL
LIN {X 0,Y 552.132,Z 282.337,A -85,B 0,C 180,E1 -3260.101,E2 -3260.101} C_VEL
LIN {X 0,Y 552.091,Z 282.336,A -85,B 0,C 180,E1 -3262.451,E2 -3262.451} C_VEL
LIN {X 0,Y 552.081,Z 282.341,A -85,B 0,C 180,E1 -3265.334,E2 -3265.334} C_VEL
LIN {X 0,Y 552.078,Z 282.339,A -85,B 0,C 180,E1 -3268.1,E2 -3268.1} C_VEL
LIN {X 0,Y 552.105,Z 282.337,A -85,B 0,C 180,E1 -3270.609,E2 -3270.609} C_VEL
LIN {X 0,Y 552.116,Z 282.336,A -85,B 0,C 180,E1 -3273.186,E2 -3273.186} C_VEL
LIN {X 0,Y 552.073,Z 282.34,A -85,B 0,C 180,E1 -3275.845,E2 -3275.845} C_VEL
LIN {X 0,Y 552.117,Z 282.335,A -85,B 0,C 180,E1 -3279.061,E2 -3279.061} C_VEL
LIN {X 0,Y 552.128,Z 282.334,A -85,B 0,C 180,E1 -3281.445,E2 -3281.445} C_VEL
LIN {X 0,Y 552.09,Z 282.336,A -85,B 0,C 180,E1 -3284.531,E2 -3284.531} C_VEL
LIN {X 0,Y 552.106,Z 282.334,A -85,B 0,C 180,E1 -3287.587,E2 -3287.587} C_VEL
LIN {X 0,Y 552.128,Z 282.338,A -85,B 0,C 180,E1 -3290.473,E2 -3290.473} C_VEL
LIN {X 0,Y 552.122,Z 282.408,A -85,B 0,C 180,E1 -3292.998,E2 -3292.998} C_VEL
LIN {X 0,Y 555.062,Z 294.146,A -85,B 0,C 180,E1 -3295.387,E2 -3295.387} C_VEL
LIN {X 0,Y 554.98,Z 300.553,A -85,B 0,C 180,E1 -3296.524,E2 -3296.524} C_VEL
LIN {X 0,Y 554.42,Z 316.967,A -85,B 0,C 180,E1 -3299.322,E2 -3299.322} C_VEL
LIN {X 0,Y 553.99,Z 335.004,A -85,B 0,C 180,E1 -3302.195,E2 -3302.195} C_VEL
LIN {X 0,Y 553.55,Z 353.043,A -85,B 0,C 180,E1 -3305.03,E2 -3305.03} C_VEL
LIN {X 0,Y 553.283,Z 370.074,A -85,B 0,C 180,E1 -3307.6,E2 -3307.6} C_VEL
LIN {X 0,Y 552.933,Z 388.662,A -85,B 0,C 180,E1 -3310.418,E2 -3310.418} C_VEL
LIN {X 0,Y 552.762,Z 396.786,A -85,B 0,C 180,E1 -3311.635,E2 -3311.635} C_VEL
LIN {X 0,Y 554.477,Z 406.014,A -85,B 0,C 180,E1 -3311.825,E2 -3311.825} C_VEL
LIN {X 0,Y 554.329,Z 421.17,A -85,B 0,C 180,E1 -3312.114,E2 -3312.114} C_VEL
LIN {X 0,Y 554.171,Z 435.294,A -85,B 0,C 180,E1 -3312.518,E2 -3312.518} C_VEL
LIN {X 0,Y 553.884,Z 449.802,A -85,B 0,C 180,E1 -3313.08,E2 -3313.08} C_VEL
LIN {X 0,Y 553.571,Z 463.882,A -85,B 0,C 180,E1 -3313.781,E2 -3313.781} C_VEL
LIN {X 0,Y 553.281,Z 477.15,A -85,B 0,C 180,E1 -3314.603,E2 -3314.603} C_VEL
LIN {X 0,Y 552.918,Z 489.864,A -85,B 0,C 180,E1 -3315.555,E2 -3315.555} C_VEL
LIN {X 0,Y 552.643,Z 501.279,A -85,B 0,C 180,E1 -3316.58,E2 -3316.58} C_VEL
LIN {X 0,Y 552.381,Z 511.766,A -85,B 0,C 180,E1 -3317.695,E2 -3317.695} C_VEL
LIN {X 0,Y 552.183,Z 522.018,A -85,B 0,C 180,E1 -3318.994,E2 -3318.994} C_VEL
LIN {X 0,Y 552.008,Z 530.535,A -85,B 0,C 180,E1 -3320.288,E2 -3320.288} C_VEL
LIN {X 0,Y 551.907,Z 537.618,A -85,B 0,C 180,E1 -3321.579,E2 -3321.579} C_VEL
LIN {X 0,Y 551.806,Z 544.186,A -85,B 0,C 180,E1 -3323.051,E2 -3323.051} C_VEL
LIN {X 0,Y 551.786,Z 549.323,A -85,B 0,C 180,E1 -3324.519,E2 -3324.519} C_VEL
LIN {X 0,Y 551.705,Z 552.291,A -85,B 0,C 180,E1 -3325.617,E2 -3325.617} C_VEL
LIN {X 0,Y 551.718,Z 555.186,A -85,B 0,C 180,E1 -3327.079,E2 -3327.079} C_VEL
LIN {X 0,Y 551.643,Z 556.911,A -85,B 0,C 180,E1 -3328.54,E2 -3328.54} C_VEL
LIN {X 0,Y 551.637,Z 557.5,A -85,B 0,C 180,E1 -3330,E2 -3330} C_VEL
LIN {X 0,Y 551.643,Z 556.909,A -85,B 0,C 180,E1 -3331.46,E2 -3331.46} C_VEL
LIN {X 0,Y 551.718,Z 555.183,A -85,B 0,C 180,E1 -3332.921,E2 -3332.921} C_VEL
LIN {X 0,Y 551.705,Z 552.289,A -85,B 0,C 180,E1 -3334.384,E2 -3334.384} C_VEL
LIN {X 0,Y 551.796,Z 548.164,A -85,B 0,C 180,E1 -3335.848,E2 -3335.848} C_VEL
LIN {X 0,Y 551.82,Z 542.701,A -85,B 0,C 180,E1 -3337.317,E2 -3337.317} C_VEL
LIN {X 0,Y 551.919,Z 535.745,A -85,B 0,C 180,E1 -3338.79,E2 -3338.79} C_VEL
LIN {X 0,Y 552.07,Z 528.291,A -85,B 0,C 180,E1 -3340.081,E2 -3340.081} C_VEL
LIN {X 0,Y 552.198,Z 519.664,A -85,B 0,C 180,E1 -3341.328,E2 -3341.328} C_VEL
LIN {X 0,Y 552.42,Z 510.136,A -85,B 0,C 180,E1 -3342.491,E2 -3342.491} C_VEL
LIN {X 0,Y 552.679,Z 499.331,A -85,B 0,C 180,E1 -3343.607,E2 -3343.607} C_VEL
LIN {X 0,Y 552.976,Z 487.532,A -85,B 0,C 180,E1 -3344.632,E2 -3344.632} C_VEL
LIN {X 0,Y 553.31,Z 474.623,A -85,B 0,C 180,E1 -3345.565,E2 -3345.565} C_VEL
LIN {X 0,Y 553.66,Z 460.355,A -85,B 0,C 180,E1 -3346.406,E2 -3346.406} C_VEL
LIN {X 0,Y 553.948,Z 446.425,A -85,B 0,C 180,E1 -3347.061,E2 -3347.061} C_VEL
LIN {X 0,Y 554.207,Z 431.531,A -85,B 0,C 180,E1 -3347.6,E2 -3347.6} C_VEL
LIN {X 0,Y 554.386,Z 416.336,A -85,B 0,C 180,E1 -3347.993,E2 -3347.993} C_VEL
LIN {X 0,Y 554.335,Z 404.812,A -85,B 0,C 180,E1 -3348.199,E2 -3348.199} C_VEL
LIN {X 0,Y 552.762,Z 396.784,A -85,B 0,C 180,E1 -3348.366,E2 -3348.366} C_VEL
LIN {X 0,Y 553.068,Z 379.029,A -85,B 0,C 180,E1 -3351.038,E2 -3351.038} C_VEL
LIN {X 0,Y 553.468,Z 360.21,A -85,B 0,C 180,E1 -3353.899,E2 -3353.899} C_VEL
LIN {X 0,Y 553.732,Z 342.434,A -85,B 0,C 180,E1 -3356.577,E2 -3356.577} C_VEL
LIN {X 0,Y 554.026,Z 325.217,A -85,B 0,C 180,E1 -3359.234,E2 -3359.234} C_VEL
LIN {X 0,Y 554.605,Z 309.594,A -85,B 0,C 180,E1 -3361.894,E2 -3361.894} C_VEL
LIN {X 0,Y 555.438,Z 298.299,A -85,B 0,C 180,E1 -3364.049,E2 -3364.049} C_VEL
LIN {X 0,Y 555.48,Z 295.217,A -85,B 0,C 180,E1 -3364.705,E2 -3364.705} C_VEL
LIN {X 0,Y 553.582,Z 287.982,A -85,B 0,C 180,E1 -3366.633,E2 -3366.633} C_VEL
LIN {X 0,Y 552.115,Z 282.339,A -85,B 0,C 180,E1 -3368.541,E2 -3368.541} C_VEL
LIN {X 0,Y 552.122,Z 282.338,A -85,B 0,C 180,E1 -3371.446,E2 -3371.446} C_VEL
LIN {X 0,Y 552.092,Z 282.341,A -85,B 0,C 180,E1 -3374.531,E2 -3374.531} C_VEL
LIN {X 0,Y 552.132,Z 282.337,A -85,B 0,C 180,E1 -3377.585,E2 -3377.585} C_VEL
LIN {X 0,Y 552.131,Z 282.338,A -85,B 0,C 180,E1 -3380.473,E2 -3380.473} C_VEL
LIN {X 0,Y 552.104,Z 282.342,A -85,B 0,C 180,E1 -3383.318,E2 -3383.318} C_VEL
LIN {X 0,Y 552.252,Z 285.258,A -85,B 0,C 180,E1 -3385.948,E2 -3385.948} C_VEL
LIN {X 0,Y 552.198,Z 287.969,A -85,B 0,C 180,E1 -3388.546,E2 -3388.546} C_VEL
LIN {X 0,Y 552.22,Z 290.688,A -85,B 0,C 180,E1 -3391.421,E2 -3391.421} C_VEL
LIN {X 0,Y 552.099,Z 293.576,A -85,B 0,C 180,E1 -3394.663,E2 -3394.663} C_VEL
LIN {X 0,Y 552.041,Z 295.381,A -85,B 0,C 180,E1 -3396.755,E2 -3396.755} C_VEL
LIN {X 0,Y 551.969,Z 297.383,A -85,B 0,C 180,E1 -3399.114,E2 -3399.114} C_VEL
LIN {X 0,Y 551.86,Z 299.411,A -85,B 0,C 180,E1 -3401.435,E2 -3401.435} C_VEL
LIN {X 0,Y 551.761,Z 301.275,A -85,B 0,C 180,E1 -3403.727,E2 -3403.727} C_VEL
LIN {X 0,Y 551.699,Z 303.25,A -85,B 0,C 180,E1 -3405.993,E2 -3405.993} C_VEL
LIN {X 0,Y 551.673,Z 304.335,A -85,B 0,C 180,E1 -3407.095,E2 -3407.095} C_VEL
LIN {X 0,Y 553.063,Z 313.668,A -85,B 0,C 180,E1 -3407.361,E2 -3407.361} C_VEL
LIN {X 0,Y 552.868,Z 326.65,A -85,B 0,C 180,E1 -3407.799,E2 -3407.799} C_VEL
LIN {X 0,Y 552.707,Z 338.615,A -85,B 0,C 180,E1 -3408.356,E2 -3408.356} C_VEL
LIN {X 0,Y 552.551,Z 349.41,A -85,B 0,C 180,E1 -3409.001,E2 -3409.001} C_VEL
LIN {X 0,Y 552.309,Z 360.449,A -85,B 0,C 180,E1 -3409.831,E2 -3409.831} C_VEL
LIN {X 0,Y 552.153,Z 371.181,A -85,B 0,C 180,E1 -3410.845,E2 -3410.845} C_VEL
LIN {X 0,Y 552.007,Z 379.101,A -85,B 0,C 180,E1 -3411.765,E2 -3411.765} C_VEL
LIN {X 0,Y 551.895,Z 386.958,A -85,B 0,C 180,E1 -3412.886,E2 -3412.886} C_VEL
LIN {X 0,Y 551.868,Z 393.956,A -85,B 0,C 180,E1 -3414.153,E2 -3414.153} C_VEL
LIN {X 0,Y 551.725,Z 398.698,A -85,B 0,C 180,E1 -3415.251,E2 -3415.251} C_VEL
LIN {X 0,Y 551.751,Z 402.329,A -85,B 0,C 180,E1 -3416.349,E2 -3416.349} C_VEL
LIN {X 0,Y 551.724,Z 404.205,A -85,B 0,C 180,E1 -3417.079,E2 -3417.079} C_VEL
LIN {X 0,Y 551.656,Z 405.626,A -85,B 0,C 180,E1 -3417.81,E2 -3417.81} C_VEL
LIN {X 0,Y 551.642,Z 407.257,A -85,B 0,C 180,E1 -3419.27,E2 -3419.27} C_VEL
LIN {X 0,Y 551.641,Z 407.496,A -85,B 0,C 180,E1 -3420,E2 -3420} C_VEL
LIN {X 0,Y 551.641,Z 407.315,A -85,B 0,C 180,E1 -3420.73,E2 -3420.73} C_VEL
LIN {X 0,Y 551.655,Z 405.768,A -85,B 0,C 180,E1 -3422.19,E2 -3422.19} C_VEL
LIN {X 0,Y 551.724,Z 404.407,A -85,B 0,C 180,E1 -3422.921,E2 -3422.921} C_VEL
LIN {X 0,Y 551.764,Z 401.525,A -85,B 0,C 180,E1 -3424.017,E2 -3424.017} C_VEL
LIN {X 0,Y 551.723,Z 397.624,A -85,B 0,C 180,E1 -3425.116,E2 -3425.116} C_VEL
LIN {X 0,Y 551.811,Z 391.893,A -85,B 0,C 180,E1 -3426.349,E2 -3426.349} C_VEL
LIN {X 0,Y 551.925,Z 385.035,A -85,B 0,C 180,E1 -3427.5,E2 -3427.5} C_VEL
LIN {X 0,Y 552.063,Z 376.856,A -85,B 0,C 180,E1 -3428.603,E2 -3428.603} C_VEL
LIN {X 0,Y 552.197,Z 368.484,A -85,B 0,C 180,E1 -3429.524,E2 -3429.524} C_VEL
LIN {X 0,Y 552.402,Z 358.156,A -85,B 0,C 180,E1 -3430.445,E2 -3430.445} C_VEL
LIN {X 0,Y 552.575,Z 346.379,A -85,B 0,C 180,E1 -3431.286,E2 -3431.286} C_VEL
LIN {X 0,Y 552.752,Z 334.944,A -85,B 0,C 180,E1 -3431.924,E2 -3431.924} C_VEL
LIN {X 0,Y 552.911,Z 322.92,A -85,B 0,C 180,E1 -3432.433,E2 -3432.433} C_VEL
LIN {X 0,Y 552.906,Z 311.692,A -85,B 0,C 180,E1 -3432.783,E2 -3432.783} C_VEL
LIN {X 0,Y 551.671,Z 304.33,A -85,B 0,C 180,E1 -3432.999,E2 -3432.999} C_VEL
LIN {X 0,Y 551.684,Z 301.608,A -85,B 0,C 180,E1 -3435.517,E2 -3435.517} C_VEL
LIN {X 0,Y 551.711,Z 299.305,A -85,B 0,C 180,E1 -3437.802,E2 -3437.802} C_VEL
LIN {X 0,Y 551.762,Z 296.849,A -85,B 0,C 180,E1 -3440.115,E2 -3440.115} C_VEL
LIN {X 0,Y 551.752,Z 294.297,A -85,B 0,C 180,E1 -3442.466,E2 -3442.466} C_VEL
LIN {X 0,Y 551.839,Z 291.334,A -85,B 0,C 180,E1 -3445.28,E2 -3445.28} C_VEL
LIN {X 0,Y 551.871,Z 288.354,A -85,B 0,C 180,E1 -3448.112,E2 -3448.112} C_VEL
LIN {X 0,Y 551.9,Z 286.53,A -85,B 0,C 180,E1 -3449.838,E2 -3449.838} C_VEL
LIN {X 0,Y 551.199,Z 285.916,A -85,B 0,C 180,E1 -3450.443,E2 -3450.443} C_VEL
LIN {X 0,Y 548.307,Z 285.049,A -85,B 0,C 180,E1 -3451.427,E2 -3451.427} C_VEL
LIN {X 0,Y 545.884,Z 284.392,A -85,B 0,C 180,E1 -3452.22,E2 -3452.22} C_VEL
LIN {X 0,Y 544.856,Z 283.821,A -85,B 0,C 180,E1 -3452.832,E2 -3452.832} C_VEL
LIN {X 0,Y 544.777,Z 283.618,A -85,B 0,C 180,E1 -3453.04,E2 -3453.04} C_VEL
LIN {X 0,Y 544.923,Z 283.235,A -85,B 0,C 180,E1 -3454.368,E2 -3454.368} C_VEL
LIN {X 0,Y 545.039,Z 283.22,A -85,B 0,C 180,E1 -3457.304,E2 -3457.304} C_VEL
LIN {X 0,Y 545.072,Z 283.21,A -85,B 0,C 180,E1 -3460.142,E2 -3460.142} C_VEL
LIN {X 0,Y 545.081,Z 283.209,A -85,B 0,C 180,E1 -3463.106,E2 -3463.106} C_VEL
LIN {X 0,Y 545.047,Z 283.22,A -85,B 0,C 180,E1 -3466.227,E2 -3466.227} C_VEL
LIN {X 0,Y 544.996,Z 283.222,A -85,B 0,C 180,E1 -3468.877,E2 -3468.877} C_VEL
LIN {X 0,Y 544.977,Z 283.433,A -85,B 0,C 180,E1 -3469.849,E2 -3469.849} C_VEL
LIN {X 0,Y 545.021,Z 286.725,A -85,B 0,C 180,E1 -3471.868,E2 -3471.868} C_VEL
LIN {X 0,Y 544.968,Z 290.711,A -85,B 0,C 180,E1 -3474.526,E2 -3474.526} C_VEL
LIN {X 0,Y 544.944,Z 294.494,A -85,B 0,C 180,E1 -3477.203,E2 -3477.203} C_VEL
LIN {X 0,Y 544.876,Z 298.089,A -85,B 0,C 180,E1 -3479.799,E2 -3479.799} C_VEL
LIN {X 0,Y 544.831,Z 301.703,A -85,B 0,C 180,E1 -3482.33,E2 -3482.33} C_VEL
LIN {X 0,Y 544.824,Z 305.238,A -85,B 0,C 180,E1 -3484.806,E2 -3484.806} C_VEL
LIN {X 0,Y 544.749,Z 308.632,A -85,B 0,C 180,E1 -3487.229,E2 -3487.229} C_VEL
LIN {X 0,Y 544.736,Z 312.95,A -85,B 0,C 180,E1 -3490.4,E2 -3490.4} C_VEL
LIN {X 0,Y 544.649,Z 314.655,A -85,B 0,C 180,E1 -3491.509,E2 -3491.509} C_VEL
LIN {X 0,Y 547.688,Z 326.937,A -85,B 0,C 180,E1 -3491.834,E2 -3491.834} C_VEL
LIN {X 0,Y 547.438,Z 341.904,A -85,B 0,C 180,E1 -3492.236,E2 -3492.236} C_VEL
LIN {X 0,Y 547.177,Z 354.147,A -85,B 0,C 180,E1 -3492.675,E2 -3492.675} C_VEL
LIN {X 0,Y 546.916,Z 365.708,A -85,B 0,C 180,E1 -3493.194,E2 -3493.194} C_VEL
LIN {X 0,Y 546.648,Z 376.248,A -85,B 0,C 180,E1 -3493.762,E2 -3493.762} C_VEL
LIN {X 0,Y 546.371,Z 386.584,A -85,B 0,C 180,E1 -3494.416,E2 -3494.416} C_VEL
LIN {X 0,Y 546.097,Z 396.903,A -85,B 0,C 180,E1 -3495.18,E2 -3495.18} C_VEL
LIN {X 0,Y 545.784,Z 406.796,A -85,B 0,C 180,E1 -3496.028,E2 -3496.028} C_VEL
LIN {X 0,Y 545.551,Z 416.269,A -85,B 0,C 180,E1 -3496.971,E2 -3496.971} C_VEL
LIN {X 0,Y 545.275,Z 426.039,A -85,B 0,C 180,E1 -3498.099,E2 -3498.099} C_VEL
LIN {X 0,Y 545.094,Z 435.588,A -85,B 0,C 180,E1 -3499.413,E2 -3499.413} C_VEL
LIN {X 0,Y 544.901,Z 443.458,A -85,B 0,C 180,E1 -3500.722,E2 -3500.722} C_VEL
LIN {X 0,Y 544.821,Z 449.173,A -85,B 0,C 180,E1 -3501.842,E2 -3501.842} C_VEL
LIN {X 0,Y 544.729,Z 453.992,A -85,B 0,C 180,E1 -3502.96,E2 -3502.96} C_VEL
LIN {X 0,Y 544.703,Z 458.018,A -85,B 0,C 180,E1 -3504.075,E2 -3504.075} C_VEL
LIN {X 0,Y 544.605,Z 462.152,A -85,B 0,C 180,E1 -3505.559,E2 -3505.559} C_VEL
LIN {X 0,Y 544.645,Z 463.824,A -85,B 0,C 180,E1 -3506.301,E2 -3506.301} C_VEL
LIN {X 0,Y 544.569,Z 466.132,A -85,B 0,C 180,E1 -3507.781,E2 -3507.781} C_VEL
LIN {X 0,Y 544.537,Z 467.283,A -85,B 0,C 180,E1 -3509.26,E2 -3509.26} C_VEL
LIN {X 0,Y 544.539,Z 467.496,A -85,B 0,C 180,E1 -3510,E2 -3510} C_VEL
LIN {X 0,Y 544.545,Z 466.955,A -85,B 0,C 180,E1 -3511.479,E2 -3511.479} C_VEL
LIN {X 0,Y 544.645,Z 465.242,A -85,B 0,C 180,E1 -3512.958,E2 -3512.958} C_VEL
LIN {X 0,Y 544.646,Z 463.999,A -85,B 0,C 180,E1 -3513.699,E2 -3513.699} C_VEL
LIN {X 0,Y 544.714,Z 459.42,A -85,B 0,C 180,E1 -3515.553,E2 -3515.553} C_VEL
LIN {X 0,Y 544.725,Z 454.332,A -85,B 0,C 180,E1 -3517.04,E2 -3517.04} C_VEL
LIN {X 0,Y 544.824,Z 447.862,A -85,B 0,C 180,E1 -3518.531,E2 -3518.531} C_VEL
LIN {X 0,Y 544.981,Z 439.666,A -85,B 0,C 180,E1 -3520.026,E2 -3520.026} C_VEL
LIN {X 0,Y 545.11,Z 432.291,A -85,B 0,C 180,E1 -3521.151,E2 -3521.151} C_VEL
LIN {X 0,Y 545.328,Z 423.673,A -85,B 0,C 180,E1 -3522.277,E2 -3522.277} C_VEL
LIN {X 0,Y 545.558,Z 415.334,A -85,B 0,C 180,E1 -3523.218,E2 -3523.218} C_VEL
LIN {X 0,Y 545.87,Z 404.694,A -85,B 0,C 180,E1 -3524.254,E2 -3524.254} C_VEL
LIN {X 0,Y 546.266,Z 391.425,A -85,B 0,C 180,E1 -3525.338,E2 -3525.338} C_VEL
LIN {X 0,Y 546.564,Z 379.36,A -85,B 0,C 180,E1 -3526.145,E2 -3526.145} C_VEL
LIN {X 0,Y 546.865,Z 367.497,A -85,B 0,C 180,E1 -3526.807,E2 -3526.807} C_VEL
LIN {X 0,Y 547.152,Z 355.888,A -85,B 0,C 180,E1 -3527.343,E2 -3527.343} C_VEL
LIN {X 0,Y 547.386,Z 343.462,A -85,B 0,C 180,E1 -3527.804,E2 -3527.804} C_VEL
LIN {X 0,Y 547.61,Z 331.162,A -85,B 0,C 180,E1 -3528.152,E2 -3528.152} C_VEL
LIN {X 0,Y 547.486,Z 326.066,A -85,B 0,C 180,E1 -3528.282,E2 -3528.282} C_VEL
LIN {X 0,Y 544.636,Z 314.476,A -85,B 0,C 180,E1 -3528.59,E2 -3528.59} C_VEL
LIN {X 0,Y 544.697,Z 312.048,A -85,B 0,C 180,E1 -3530.388,E2 -3530.388} C_VEL
LIN {X 0,Y 544.748,Z 308.799,A -85,B 0,C 180,E1 -3532.77,E2 -3532.77} C_VEL
LIN {X 0,Y 544.806,Z 305.022,A -85,B 0,C 180,E1 -3535.445,E2 -3535.445} C_VEL
LIN {X 0,Y 544.926,Z 300.623,A -85,B 0,C 180,E1 -3538.502,E2 -3538.502} C_VEL
LIN {X 0,Y 544.929,Z 296.184,A -85,B 0,C 180,E1 -3541.657,E2 -3541.657} C_VEL
LIN {X 0,Y 544.967,Z 292.151,A -85,B 0,C 180,E1 -3544.571,E2 -3544.571} C_VEL
LIN {X 0,Y 544.989,Z 288.154,A -85,B 0,C 180,E1 -3547.308,E2 -3547.308} C_VEL
LIN {X 0,Y 544.99,Z 283.59,A -85,B 0,C 180,E1 -3550.149,E2 -3550.149} C_VEL
LIN {X 0,Y 544.989,Z 283.232,A -85,B 0,C 180,E1 -3550.461,E2 -3550.461} C_VEL
LIN {X 0,Y 545.045,Z 283.217,A -85,B 0,C 180,E1 -3553.11,E2 -3553.11} C_VEL
LIN {X 0,Y 545.05,Z 283.215,A -85,B 0,C 180,E1 -3556.226,E2 -3556.226} C_VEL
LIN {X 0,Y 545.081,Z 283.214,A -85,B 0,C 180,E1 -3558.885,E2 -3558.885} C_VEL
LIN {X 0,Y 545.042,Z 283.22,A -85,B 0,C 180,E1 -3561.865,E2 -3561.865} C_VEL
LIN {X 0,Y 545.046,Z 283.215,A -85,B 0,C 180,E1 -3564.532,E2 -3564.532} C_VEL
LIN {X 0,Y 545.069,Z 283.215,A -85,B 0,C 180,E1 -3567.211,E2 -3567.211} C_VEL
LIN {X 0,Y 545.062,Z 283.213,A -85,B 0,C 180,E1 -3569.81,E2 -3569.81} C_VEL
LIN {X 0,Y 545.023,Z 283.217,A -85,B 0,C 180,E1 -3572.841,E2 -3572.841} C_VEL
LIN {X 0,Y 545.046,Z 283.217,A -85,B 0,C 180,E1 -3575.63,E2 -3575.63} C_VEL
LIN {X 0,Y 545.065,Z 283.215,A -85,B 0,C 180,E1 -3578.837,E2 -3578.837} C_VEL
LIN {X 0,Y 545.048,Z 283.214,A -85,B 0,C 180,E1 -3581.194,E2 -3581.194} C_VEL
LIN {X 0,Y 545.038,Z 283.217,A -85,B 0,C 180,E1 -3583.52,E2 -3583.52} C_VEL
LIN {X 0,Y 545.096,Z 283.209,A -85,B 0,C 180,E1 -3585.82,E2 -3585.82} C_VEL
LIN {X 0,Y 545.12,Z 283.207,A -85,B 0,C 180,E1 -3588.849,E2 -3588.849} C_VEL
LIN {X 0,Y 545.085,Z 283.215,A -85,B 0,C 180,E1 -3591.846,E2 -3591.846} C_VEL
LIN {X 0,Y 545.192,Z 283.194,A -85,B 0,C 180,E1 -3594.823,E2 -3594.823} C_VEL
LIN {X 0,Y 545.193,Z 283.196,A -85,B 0,C 180,E1 -3597.784,E2 -3597.784} C_VEL
LIN {X 0,Y 545.21,Z 283.194,A -85,B 0,C 180,E1 -3600.739,E2 -3600.739} C_VEL
LIN {X 0,Y 545.158,Z 283.201,A -85,B 0,C 180,E1 -3602.956,E2 -3602.956} C_VEL
LIN {X 0,Y 545.132,Z 283.201,A -85,B 0,C 180,E1 -3605.92,E2 -3605.92} C_VEL
LIN {X 0,Y 545.111,Z 283.208,A -85,B 0,C 180,E1 -3608.9,E2 -3608.9} C_VEL
LIN {X 0,Y 545.105,Z 283.209,A -85,B 0,C 180,E1 -3611.905,E2 -3611.905} C_VEL
LIN {X 0,Y 545.076,Z 283.213,A -85,B 0,C 180,E1 -3614.944,E2 -3614.944} C_VEL
LIN {X 0,Y 545.069,Z 283.211,A -85,B 0,C 180,E1 -3618.026,E2 -3618.026} C_VEL
LIN {X 0,Y 545.096,Z 283.211,A -85,B 0,C 180,E1 -3620.372,E2 -3620.372} C_VEL
LIN {X 0,Y 545.073,Z 283.217,A -85,B 0,C 180,E1 -3623.56,E2 -3623.56} C_VEL
LIN {X 0,Y 545.045,Z 283.212,A -85,B 0,C 180,E1 -3626.002,E2 -3626.002} C_VEL
LIN {X 0,Y 545.07,Z 283.216,A -85,B 0,C 180,E1 -3628.744,E2 -3628.744} C_VEL
LIN {X 0,Y 545.058,Z 283.217,A -85,B 0,C 180,E1 -3631.679,E2 -3631.679} C_VEL
LIN {X 0,Y 545.061,Z 283.213,A -85,B 0,C 180,E1 -3634.564,E2 -3634.564} C_VEL
LIN {X 0,Y 545.025,Z 283.219,A -85,B 0,C 180,E1 -3637.305,E2 -3637.305} C_VEL
LIN {X 0,Y 545.064,Z 283.218,A -85,B 0,C 180,E1 -3640.143,E2 -3640.143} C_VEL
LIN {X 0,Y 545.078,Z 283.211,A -85,B 0,C 180,E1 -3643.107,E2 -3643.107} C_VEL
LIN {X 0,Y 545.048,Z 283.213,A -85,B 0,C 180,E1 -3646.226,E2 -3646.226} C_VEL
LIN {X 0,Y 545.027,Z 283.22,A -85,B 0,C 180,E1 -3648.88,E2 -3648.88} C_VEL
LIN {X 0,Y 545.079,Z 283.215,A -85,B 0,C 180,E1 -3650.818,E2 -3650.818} C_VEL
LIN {X 0,Y 545.068,Z 283.258,A -85,B 0,C 180,E1 -3652.583,E2 -3652.583} C_VEL
LIN {X 0,Y 548.371,Z 296.292,A -85,B 0,C 180,E1 -3655.295,E2 -3655.295} C_VEL
LIN {X 0,Y 548.153,Z 305.757,A -85,B 0,C 180,E1 -3656.982,E2 -3656.982} C_VEL
LIN {X 0,Y 547.501,Z 321.23,A -85,B 0,C 180,E1 -3659.627,E2 -3659.627} C_VEL
LIN {X 0,Y 547.076,Z 337.511,A -85,B 0,C 180,E1 -3662.267,E2 -3662.267} C_VEL
LIN {X 0,Y 546.606,Z 355.225,A -85,B 0,C 180,E1 -3665.097,E2 -3665.097} C_VEL
LIN {X 0,Y 546.299,Z 373.569,A -85,B 0,C 180,E1 -3667.859,E2 -3667.859} C_VEL
LIN {X 0,Y 545.938,Z 390.547,A -85,B 0,C 180,E1 -3670.446,E2 -3670.446} C_VEL
LIN {X 0,Y 545.803,Z 396.809,A -85,B 0,C 180,E1 -3671.396,E2 -3671.396} C_VEL
LIN {X 0,Y 547.741,Z 407.048,A -85,B 0,C 180,E1 -3671.61,E2 -3671.61} C_VEL
LIN {X 0,Y 547.559,Z 422.32,A -85,B 0,C 180,E1 -3671.915,E2 -3671.915} C_VEL
LIN {X 0,Y 547.363,Z 436.629,A -85,B 0,C 180,E1 -3672.343,E2 -3672.343} C_VEL
LIN {X 0,Y 547.045,Z 450.828,A -85,B 0,C 180,E1 -3672.91,E2 -3672.91} C_VEL
LIN {X 0,Y 546.671,Z 465.517,A -85,B 0,C 180,E1 -3673.667,E2 -3673.667} C_VEL
LIN {X 0,Y 546.373,Z 478.415,A -85,B 0,C 180,E1 -3674.491,E2 -3674.491} C_VEL
LIN {X 0,Y 545.958,Z 491.014,A -85,B 0,C 180,E1 -3675.462,E2 -3675.462} C_VEL
LIN {X 0,Y 545.639,Z 503.188,A -85,B 0,C 180,E1 -3676.594,E2 -3676.594} C_VEL
LIN {X 0,Y 545.357,Z 513.391,A -85,B 0,C 180,E1 -3677.723,E2 -3677.723} C_VEL
LIN {X 0,Y 545.155,Z 523.368,A -85,B 0,C 180,E1 -3679.038,E2 -3679.038} C_VEL
LIN {X 0,Y 544.904,Z 531.649,A -85,B 0,C 180,E1 -3680.348,E2 -3680.348} C_VEL
LIN {X 0,Y 544.818,Z 539.423,A -85,B 0,C 180,E1 -3681.843,E2 -3681.843} C_VEL
LIN {X 0,Y 544.704,Z 546.08,A -85,B 0,C 180,E1 -3683.456,E2 -3683.456} C_VEL
LIN {X 0,Y 544.642,Z 550.385,A -85,B 0,C 180,E1 -3684.818,E2 -3684.818} C_VEL
LIN {X 0,Y 544.644,Z 553.888,A -85,B 0,C 180,E1 -3686.301,E2 -3686.301} C_VEL
LIN {X 0,Y 544.569,Z 556.191,A -85,B 0,C 180,E1 -3687.781,E2 -3687.781} C_VEL
LIN {X 0,Y 544.539,Z 557.349,A -85,B 0,C 180,E1 -3689.261,E2 -3689.261} C_VEL
LIN {X 0,Y 544.539,Z 557.348,A -85,B 0,C 180,E1 -3690.74,E2 -3690.74} C_VEL
LIN {X 0,Y 544.569,Z 556.188,A -85,B 0,C 180,E1 -3692.219,E2 -3692.219} C_VEL
LIN {X 0,Y 544.644,Z 553.885,A -85,B 0,C 180,E1 -3693.699,E2 -3693.699} C_VEL
LIN {X 0,Y 544.642,Z 550.386,A -85,B 0,C 180,E1 -3695.183,E2 -3695.183} C_VEL
LIN {X 0,Y 544.752,Z 545.608,A -85,B 0,C 180,E1 -3696.668,E2 -3696.668} C_VEL
LIN {X 0,Y 544.819,Z 539.42,A -85,B 0,C 180,E1 -3698.158,E2 -3698.158} C_VEL
LIN {X 0,Y 544.904,Z 531.644,A -85,B 0,C 180,E1 -3699.653,E2 -3699.653} C_VEL
LIN {X 0,Y 545.15,Z 523.366,A -85,B 0,C 180,E1 -3700.962,E2 -3700.962} C_VEL
LIN {X 0,Y 545.358,Z 513.39,A -85,B 0,C 180,E1 -3702.277,E2 -3702.277} C_VEL
LIN {X 0,Y 545.639,Z 503.184,A -85,B 0,C 180,E1 -3703.406,E2 -3703.406} C_VEL
LIN {X 0,Y 545.971,Z 491.016,A -85,B 0,C 180,E1 -3704.538,E2 -3704.538} C_VEL
LIN {X 0,Y 546.355,Z 478.641,A -85,B 0,C 180,E1 -3705.493,E2 -3705.493} C_VEL
LIN {X 0,Y 546.684,Z 465.504,A -85,B 0,C 180,E1 -3706.333,E2 -3706.333} C_VEL
LIN {X 0,Y 547.034,Z 450.82,A -85,B 0,C 180,E1 -3707.091,E2 -3707.091} C_VEL
LIN {X 0,Y 547.379,Z 435.346,A -85,B 0,C 180,E1 -3707.705,E2 -3707.705} C_VEL
LIN {X 0,Y 547.619,Z 419.66,A -85,B 0,C 180,E1 -3708.152,E2 -3708.152} C_VEL
LIN {X 0,Y 547.549,Z 405.431,A -85,B 0,C 180,E1 -3708.422,E2 -3708.422} C_VEL
LIN {X 0,Y 545.799,Z 396.784,A -85,B 0,C 180,E1 -3708.608,E2 -3708.608} C_VEL
LIN {X 0,Y 546.199,Z 379.029,A -85,B 0,C 180,E1 -3711.315,E2 -3711.315} C_VEL
LIN {X 0,Y 546.427,Z 362.294,A -85,B 0,C 180,E1 -3713.777,E2 -3713.777} C_VEL
LIN {X 0,Y 546.771,Z 342.982,A -85,B 0,C 180,E1 -3716.736,E2 -3716.736} C_VEL
LIN {X 0,Y 547.125,Z 327.353,A -85,B 0,C 180,E1 -3719.218,E2 -3719.218} C_VEL
LIN {X 0,Y 547.723,Z 312.808,A -85,B 0,C 180,E1 -3721.741,E2 -3721.741} C_VEL
LIN {X 0,Y 548.566,Z 301.671,A -85,B 0,C 180,E1 -3723.884,E2 -3723.884} C_VEL
LIN {X 0,Y 548.838,Z 298.281,A -85,B 0,C 180,E1 -3724.604,E2 -3724.604} C_VEL
LIN {X 0,Y 547.44,Z 292.18,A -85,B 0,C 180,E1 -3726.196,E2 -3726.196} C_VEL
LIN {X 0,Y 545.709,Z 285.934,A -85,B 0,C 180,E1 -3728.224,E2 -3728.224} C_VEL
LIN {X 0,Y 545.088,Z 283.214,A -85,B 0,C 180,E1 -3729.369,E2 -3729.369} C_VEL
LIN {X 0,Y 545.079,Z 283.216,A -85,B 0,C 180,E1 -3732.103,E2 -3732.103} C_VEL
LIN {X 0,Y 545.036,Z 283.221,A -85,B 0,C 180,E1 -3734.83,E2 -3734.83} C_VEL
LIN {X 0,Y 545.08,Z 283.216,A -85,B 0,C 180,E1 -3737.897,E2 -3737.897} C_VEL
LIN {X 0,Y 545.082,Z 283.216,A -85,B 0,C 180,E1 -3740.819,E2 -3740.819} C_VEL
LIN {X 0,Y 545.095,Z 283.445,A -85,B 0,C 180,E1 -3743.071,E2 -3743.071} C_VEL
LIN {X 0,Y 545.26,Z 286.13,A -85,B 0,C 180,E1 -3745.58,E2 -3745.58} C_VEL
LIN {X 0,Y 545.201,Z 288.908,A -85,B 0,C 180,E1 -3748.298,E2 -3748.298} C_VEL
LIN {X 0,Y 545.193,Z 291.643,A -85,B 0,C 180,E1 -3751.233,E2 -3751.233} C_VEL
LIN {X 0,Y 545.101,Z 294.112,A -85,B 0,C 180,E1 -3754.001,E2 -3754.001} C_VEL
LIN {X 0,Y 545.062,Z 296.209,A -85,B 0,C 180,E1 -3756.44,E2 -3756.44} C_VEL
LIN {X 0,Y 544.922,Z 298.929,A -85,B 0,C 180,E1 -3759.621,E2 -3759.621} C_VEL
LIN {X 0,Y 544.807,Z 300.969,A -85,B 0,C 180,E1 -3761.965,E2 -3761.965} C_VEL
LIN {X 0,Y 544.722,Z 302.858,A -85,B 0,C 180,E1 -3764.28,E2 -3764.28} C_VEL
LIN {X 0,Y 544.677,Z 305.332,A -85,B 0,C 180,E1 -3766.92,E2 -3766.92} C_VEL
LIN {X 0,Y 546.204,Z 314.723,A -85,B 0,C 180,E1 -3767.2,E2 -3767.2} C_VEL
LIN {X 0,Y 545.989,Z 327.356,A -85,B 0,C 180,E1 -3767.643,E2 -3767.643} C_VEL
LIN {X 0,Y 545.773,Z 339.295,A -85,B 0,C 180,E1 -3768.218,E2 -3768.218} C_VEL
LIN {X 0,Y 545.546,Z 351.018,A -85,B 0,C 180,E1 -3768.952,E2 -3768.952} C_VEL
LIN {X 0,Y 545.29,Z 361.558,A -85,B 0,C 180,E1 -3769.792,E2 -3769.792} C_VEL
LIN {X 0,Y 545.122,Z 371.185,A -85,B 0,C 180,E1 -3770.726,E2 -3770.726} C_VEL
LIN {X 0,Y 544.975,Z 379.105,A -85,B 0,C 180,E1 -3771.658,E2 -3771.658} C_VEL
LIN {X 0,Y 544.83,Z 386.849,A -85,B 0,C 180,E1 -3772.775,E2 -3772.775} C_VEL
LIN {X 0,Y 544.778,Z 393.959,A -85,B 0,C 180,E1 -3774.076,E2 -3774.076} C_VEL
LIN {X 0,Y 544.629,Z 398.7,A -85,B 0,C 180,E1 -3775.189,E2 -3775.189} C_VEL
LIN {X 0,Y 544.669,Z 402.33,A -85,B 0,C 180,E1 -3776.301,E2 -3776.301} C_VEL
LIN {X 0,Y 544.651,Z 404.206,A -85,B 0,C 180,E1 -3777.041,E2 -3777.041} C_VEL
LIN {X 0,Y 544.57,Z 405.626,A -85,B 0,C 180,E1 -3777.781,E2 -3777.781} C_VEL
LIN {X 0,Y 544.543,Z 407.257,A -85,B 0,C 180,E1 -3779.261,E2 -3779.261} C_VEL
LIN {X 0,Y 544.541,Z 407.496,A -85,B 0,C 180,E1 -3780,E2 -3780} C_VEL
LIN {X 0,Y 544.542,Z 407.315,A -85,B 0,C 180,E1 -3780.74,E2 -3780.74} C_VEL
LIN {X 0,Y 544.57,Z 405.766,A -85,B 0,C 180,E1 -3782.219,E2 -3782.219} C_VEL
LIN {X 0,Y 544.651,Z 404.405,A -85,B 0,C 180,E1 -3782.959,E2 -3782.959} C_VEL
LIN {X 0,Y 544.684,Z 401.523,A -85,B 0,C 180,E1 -3784.07,E2 -3784.07} C_VEL
LIN {X 0,Y 544.653,Z 397.621,A -85,B 0,C 180,E1 -3785.182,E2 -3785.182} C_VEL
LIN {X 0,Y 544.725,Z 392.4,A -85,B 0,C 180,E1 -3786.335,E2 -3786.335} C_VEL
LIN {X 0,Y 544.859,Z 385.031,A -85,B 0,C 180,E1 -3787.598,E2 -3787.598} C_VEL
LIN {X 0,Y 544.999,Z 376.851,A -85,B 0,C 180,E1 -3788.715,E2 -3788.715} C_VEL
LIN {X 0,Y 545.16,Z 368.478,A -85,B 0,C 180,E1 -3789.648,E2 -3789.648} C_VEL
LIN {X 0,Y 545.381,Z 358.158,A -85,B 0,C 180,E1 -3790.581,E2 -3790.581} C_VEL
LIN {X 0,Y 545.596,Z 346.909,A -85,B 0,C 180,E1 -3791.405,E2 -3791.405} C_VEL
LIN {X 0,Y 545.818,Z 335.188,A -85,B 0,C 180,E1 -3792.078,E2 -3792.078} C_VEL
LIN {X 0,Y 545.998,Z 323.277,A -85,B 0,C 180,E1 -3792.593,E2 -3792.593} C_VEL
LIN {X 0,Y 546.02,Z 312.658,A -85,B 0,C 180,E1 -3792.935,E2 -3792.935} C_VEL
LIN {X 0,Y 544.602,Z 304.706,A -85,B 0,C 180,E1 -3793.171,E2 -3793.171} C_VEL
LIN {X 0,Y 544.625,Z 302.077,A -85,B 0,C 180,E1 -3795.723,E2 -3795.723} C_VEL
LIN {X 0,Y 544.64,Z 299.78,A -85,B 0,C 180,E1 -3798.041,E2 -3798.041} C_VEL
LIN {X 0,Y 544.706,Z 297.198,A -85,B 0,C 180,E1 -3800.387,E2 -3800.387} C_VEL
LIN {X 0,Y 544.688,Z 294.651,A -85,B 0,C 180,E1 -3802.773,E2 -3802.773} C_VEL
LIN {X 0,Y 544.774,Z 291.836,A -85,B 0,C 180,E1 -3805.437,E2 -3805.437} C_VEL
LIN {X 0,Y 544.832,Z 288.621,A -85,B 0,C 180,E1 -3808.508,E2 -3808.508} C_VEL
LIN {X 0,Y 544.766,Z 285.777,A -85,B 0,C 180,E1 -3811.067,E2 -3811.067} C_VEL
LIN {X 0,Y 544.777,Z 283.618,A -85,B 0,C 180,E1 -3813.04,E2 -3813.04} C_VEL
LIN {X 0,Y 544.138,Z 283.448,A -85,B 0,C 180,E1 -3813.658,E2 -3813.658} C_VEL
LIN {X 0,Y 541.36,Z 283.679,A -85,B 0,C 180,E1 -3814.663,E2 -3814.663} C_VEL
LIN {X 0,Y 539.018,Z 283.97,A -85,B 0,C 180,E1 -3815.472,E2 -3815.472} C_VEL
LIN {X 0,Y 538.032,Z 284.088,A -85,B 0,C 180,E1 -3816.097,E2 -3816.097} C_VEL
LIN {X 0,Y 537.962,Z 284.096,A -85,B 0,C 180,E1 -3816.308,E2 -3816.308} C_VEL
LIN {X 0,Y 538.019,Z 284.095,A -85,B 0,C 180,E1 -3818.83,E2 -3818.83} C_VEL
LIN {X 0,Y 538.033,Z 284.086,A -85,B 0,C 180,E1 -3821.773,E2 -3821.773} C_VEL
LIN {X 0,Y 538.003,Z 284.092,A -85,B 0,C 180,E1 -3824.863,E2 -3824.863} C_VEL
LIN {X 0,Y 537.989,Z 284.094,A -85,B 0,C 180,E1 -3827.211,E2 -3827.211} C_VEL
LIN {X 0,Y 537.947,Z 284.102,A -85,B 0,C 180,E1 -3829.265,E2 -3829.265} C_VEL
LIN {X 0,Y 537.957,Z 285.28,A -85,B 0,C 180,E1 -3830.425,E2 -3830.425} C_VEL
LIN {X 0,Y 537.93,Z 289.402,A -85,B 0,C 180,E1 -3833.059,E2 -3833.059} C_VEL
LIN {X 0,Y 537.897,Z 293.377,A -85,B 0,C 180,E1 -3835.818,E2 -3835.818} C_VEL
LIN {X 0,Y 537.864,Z 297.054,A -85,B 0,C 180,E1 -3838.489,E2 -3838.489} C_VEL
LIN {X 0,Y 537.807,Z 300.704,A -85,B 0,C 180,E1 -3841.11,E2 -3841.11} C_VEL
LIN {X 0,Y 537.763,Z 304.296,A -85,B 0,C 180,E1 -3843.618,E2 -3843.618} C_VEL
LIN {X 0,Y 537.713,Z 307.994,A -85,B 0,C 180,E1 -3846.193,E2 -3846.193} C_VEL
LIN {X 0,Y 537.667,Z 311.284,A -85,B 0,C 180,E1 -3848.531,E2 -3848.531} C_VEL
LIN {X 0,Y 537.627,Z 314.55,A -85,B 0,C 180,E1 -3850.925,E2 -3850.925} C_VEL
LIN {X 0,Y 537.638,Z 315.074,A -85,B 0,C 180,E1 -3851.258,E2 -3851.258} C_VEL
LIN {X 0,Y 540.927,Z 328.393,A -85,B 0,C 180,E1 -3851.63,E2 -3851.63} C_VEL
LIN {X 0,Y 540.677,Z 342.073,A -85,B 0,C 180,E1 -3852.008,E2 -3852.008} C_VEL
LIN {X 0,Y 540.393,Z 354.359,A -85,B 0,C 180,E1 -3852.459,E2 -3852.459} C_VEL
LIN {X 0,Y 540.085,Z 365.703,A -85,B 0,C 180,E1 -3852.975,E2 -3852.975} C_VEL
LIN {X 0,Y 539.805,Z 376.245,A -85,B 0,C 180,E1 -3853.55,E2 -3853.55} C_VEL
LIN {X 0,Y 539.478,Z 386.682,A -85,B 0,C 180,E1 -3854.219,E2 -3854.219} C_VEL
LIN {X 0,Y 539.195,Z 396.9,A -85,B 0,C 180,E1 -3854.986,E2 -3854.986} C_VEL
LIN {X 0,Y 538.863,Z 406.792,A -85,B 0,C 180,E1 -3855.845,E2 -3855.845} C_VEL
LIN {X 0,Y 538.582,Z 416.267,A -85,B 0,C 180,E1 -3856.799,E2 -3856.799} C_VEL
LIN {X 0,Y 538.282,Z 426.035,A -85,B 0,C 180,E1 -3857.942,E2 -3857.942} C_VEL
LIN {X 0,Y 538.069,Z 435.594,A -85,B 0,C 180,E1 -3859.273,E2 -3859.273} C_VEL
LIN {X 0,Y 537.827,Z 443.456,A -85,B 0,C 180,E1 -3860.599,E2 -3860.599} C_VEL
LIN {X 0,Y 537.736,Z 449.169,A -85,B 0,C 180,E1 -3861.734,E2 -3861.734} C_VEL
LIN {X 0,Y 537.651,Z 453.989,A -85,B 0,C 180,E1 -3862.866,E2 -3862.866} C_VEL
LIN {X 0,Y 537.641,Z 459.14,A -85,B 0,C 180,E1 -3864.374,E2 -3864.374} C_VEL
LIN {X 0,Y 537.562,Z 463.828,A -85,B 0,C 180,E1 -3866.252,E2 -3866.252} C_VEL
LIN {X 0,Y 537.488,Z 466.132,A -85,B 0,C 180,E1 -3867.752,E2 -3867.752} C_VEL
LIN {X 0,Y 537.437,Z 467.277,A -85,B 0,C 180,E1 -3869.251,E2 -3869.251} C_VEL
LIN {X 0,Y 537.44,Z 467.496,A -85,B 0,C 180,E1 -3870,E2 -3870} C_VEL
LIN {X 0,Y 537.45,Z 466.95,A -85,B 0,C 180,E1 -3871.498,E2 -3871.498} C_VEL
LIN {X 0,Y 537.545,Z 465.234,A -85,B 0,C 180,E1 -3872.998,E2 -3872.998} C_VEL
LIN {X 0,Y 537.562,Z 464.001,A -85,B 0,C 180,E1 -3873.748,E2 -3873.748} C_VEL
LIN {X 0,Y 537.641,Z 459.411,A -85,B 0,C 180,E1 -3875.626,E2 -3875.626} C_VEL
LIN {X 0,Y 537.619,Z 455.726,A -85,B 0,C 180,E1 -3876.756,E2 -3876.756} C_VEL
LIN {X 0,Y 537.695,Z 451.264,A -85,B 0,C 180,E1 -3877.888,E2 -3877.888} C_VEL
LIN {X 0,Y 537.802,Z 444.932,A -85,B 0,C 180,E1 -3879.212,E2 -3879.212} C_VEL
LIN {X 0,Y 537.995,Z 438.487,A -85,B 0,C 180,E1 -3880.348,E2 -3880.348} C_VEL
LIN {X 0,Y 538.122,Z 431.099,A -85,B 0,C 180,E1 -3881.464,E2 -3881.464} C_VEL
LIN {X 0,Y 538.368,Z 422.104,A -85,B 0,C 180,E1 -3882.63,E2 -3882.63} C_VEL
LIN {X 0,Y 538.722,Z 411.75,A -85,B 0,C 180,E1 -3883.773,E2 -3883.773} C_VEL
LIN {X 0,Y 539.112,Z 399.186,A -85,B 0,C 180,E1 -3884.92,E2 -3884.92} C_VEL
LIN {X 0,Y 539.471,Z 388.032,A -85,B 0,C 180,E1 -3885.775,E2 -3885.775} C_VEL
LIN {X 0,Y 539.773,Z 377.734,A -85,B 0,C 180,E1 -3886.451,E2 -3886.451} C_VEL
LIN {X 0,Y 540.038,Z 367.467,A -85,B 0,C 180,E1 -3887.026,E2 -3887.026} C_VEL
LIN {X 0,Y 540.294,Z 357.863,A -85,B 0,C 180,E1 -3887.485,E2 -3887.485} C_VEL
LIN {X 0,Y 540.617,Z 344.579,A -85,B 0,C 180,E1 -3887.998,E2 -3887.998} C_VEL
LIN {X 0,Y 540.856,Z 332.233,A -85,B 0,C 180,E1 -3888.364,E2 -3888.364} C_VEL
LIN {X 0,Y 540.784,Z 327.533,A -85,B 0,C 180,E1 -3888.486,E2 -3888.486} C_VEL
LIN {X 0,Y 537.624,Z 314.996,A -85,B 0,C 180,E1 -3888.847,E2 -3888.847} C_VEL
LIN {X 0,Y 537.665,Z 311.408,A -85,B 0,C 180,E1 -3891.469,E2 -3891.469} C_VEL
LIN {X 0,Y 537.723,Z 307.993,A -85,B 0,C 180,E1 -3893.902,E2 -3893.902} C_VEL
LIN {X 0,Y 537.766,Z 304.429,A -85,B 0,C 180,E1 -3896.381,E2 -3896.381} C_VEL
LIN {X 0,Y 537.86,Z 300.786,A -85,B 0,C 180,E1 -3898.912,E2 -3898.912} C_VEL
LIN {X 0,Y 537.872,Z 296.699,A -85,B 0,C 180,E1 -3901.863,E2 -3901.863} C_VEL
LIN {X 0,Y 537.913,Z 292.926,A -85,B 0,C 180,E1 -3904.602,E2 -3904.602} C_VEL
LIN {X 0,Y 537.943,Z 289.221,A -85,B 0,C 180,E1 -3907.161,E2 -3907.161} C_VEL
LIN {X 0,Y 537.953,Z 285.059,A -85,B 0,C 180,E1 -3909.803,E2 -3909.803} C_VEL
LIN {X 0,Y 537.95,Z 284.106,A -85,B 0,C 180,E1 -3910.785,E2 -3910.785} C_VEL
LIN {X 0,Y 538.011,Z 284.097,A -85,B 0,C 180,E1 -3913.815,E2 -3913.815} C_VEL
LIN {X 0,Y 538.004,Z 284.093,A -85,B 0,C 180,E1 -3916.184,E2 -3916.184} C_VEL
LIN {X 0,Y 538.048,Z 284.087,A -85,B 0,C 180,E1 -3919.253,E2 -3919.253} C_VEL
LIN {X 0,Y 537.985,Z 284.099,A -85,B 0,C 180,E1 -3922.122,E2 -3922.122} C_VEL
LIN {X 0,Y 538.009,Z 284.094,A -85,B 0,C 180,E1 -3924.916,E2 -3924.916} C_VEL
LIN {X 0,Y 538.019,Z 284.09,A -85,B 0,C 180,E1 -3927.617,E2 -3927.617} C_VEL
LIN {X 0,Y 537.997,Z 284.096,A -85,B 0,C 180,E1 -3930.238,E2 -3930.238} C_VEL
LIN {X 0,Y 537.993,Z 284.092,A -85,B 0,C 180,E1 -3932.792,E2 -3932.792} C_VEL
LIN {X 0,Y 538.017,Z 284.095,A -85,B 0,C 180,E1 -3935.291,E2 -3935.291} C_VEL
LIN {X 0,Y 538.016,Z 284.088,A -85,B 0,C 180,E1 -3938.042,E2 -3938.042} C_VEL
LIN {X 0,Y 538.081,Z 284.086,A -85,B 0,C 180,E1 -3940.148,E2 -3940.148} C_VEL
LIN {X 0,Y 537.987,Z 284.093,A -85,B 0,C 180,E1 -3943.298,E2 -3943.298} C_VEL
LIN {X 0,Y 538.065,Z 284.086,A -85,B 0,C 180,E1 -3945.631,E2 -3945.631} C_VEL
LIN {X 0,Y 538.079,Z 284.084,A -85,B 0,C 180,E1 -3948.701,E2 -3948.701} C_VEL
LIN {X 0,Y 538.052,Z 284.09,A -85,B 0,C 180,E1 -3951.739,E2 -3951.739} C_VEL
LIN {X 0,Y 538.147,Z 284.071,A -85,B 0,C 180,E1 -3954.755,E2 -3954.755} C_VEL
LIN {X 0,Y 538.165,Z 284.071,A -85,B 0,C 180,E1 -3957.755,E2 -3957.755} C_VEL
LIN {X 0,Y 538.181,Z 284.069,A -85,B 0,C 180,E1 -3960.748,E2 -3960.748} C_VEL
LIN {X 0,Y 538.126,Z 284.077,A -85,B 0,C 180,E1 -3962.994,E2 -3962.994} C_VEL
LIN {X 0,Y 538.088,Z 284.078,A -85,B 0,C 180,E1 -3965.998,E2 -3965.998} C_VEL
LIN {X 0,Y 538.064,Z 284.085,A -85,B 0,C 180,E1 -3969.018,E2 -3969.018} C_VEL
LIN {X 0,Y 538.064,Z 284.088,A -85,B 0,C 180,E1 -3972.063,E2 -3972.063} C_VEL
LIN {X 0,Y 538.038,Z 284.092,A -85,B 0,C 180,E1 -3975.144,E2 -3975.144} C_VEL
LIN {X 0,Y 538.025,Z 284.091,A -85,B 0,C 180,E1 -3978.27,E2 -3978.27} C_VEL
LIN {X 0,Y 538.04,Z 284.086,A -85,B 0,C 180,E1 -3980.651,E2 -3980.651} C_VEL
LIN {X 0,Y 537.997,Z 284.095,A -85,B 0,C 180,E1 -3983.889,E2 -3983.889} C_VEL
LIN {X 0,Y 537.992,Z 284.091,A -85,B 0,C 180,E1 -3986.369,E2 -3986.369} C_VEL
LIN {X 0,Y 538.03,Z 284.091,A -85,B 0,C 180,E1 -3988.933,E2 -3988.933} C_VEL
LIN {X 0,Y 538.011,Z 284.097,A -85,B 0,C 180,E1 -3991.887,E2 -3991.887} C_VEL
LIN {X 0,Y 538.01,Z 284.091,A -85,B 0,C 180,E1 -3994.617,E2 -3994.617} C_VEL
LIN {X 0,Y 537.995,Z 284.096,A -85,B 0,C 180,E1 -3997.169,E2 -3997.169} C_VEL
LIN {X 0,Y 538.009,Z 284.093,A -85,B 0,C 180,E1 -3999.798,E2 -3999.798} C_VEL
LIN {X 0,Y 538.019,Z 284.089,A -85,B 0,C 180,E1 -4002.786,E2 -4002.786} C_VEL
LIN {X 0,Y 538.018,Z 284.089,A -85,B 0,C 180,E1 -4005.927,E2 -4005.927} C_VEL
LIN {X 0,Y 538.001,Z 284.095,A -85,B 0,C 180,E1 -4009.22,E2 -4009.22} C_VEL
LIN {X 0,Y 538.021,Z 284.154,A -85,B 0,C 180,E1 -4012.17,E2 -4012.17} C_VEL
LIN {X 0,Y 541.29,Z 296.883,A -85,B 0,C 180,E1 -4014.883,E2 -4014.883} C_VEL
LIN {X 0,Y 541.718,Z 299.569,A -85,B 0,C 180,E1 -4015.418,E2 -4015.418} C_VEL
LIN {X 0,Y 541.199,Z 311.639,A -85,B 0,C 180,E1 -4017.574,E2 -4017.574} C_VEL
LIN {X 0,Y 540.544,Z 328.084,A -85,B 0,C 180,E1 -4020.392,E2 -4020.392} C_VEL
LIN {X 0,Y 539.983,Z 345.945,A -85,B 0,C 180,E1 -4023.319,E2 -4023.319} C_VEL
LIN {X 0,Y 539.489,Z 365.202,A -85,B 0,C 180,E1 -4026.385,E2 -4026.385} C_VEL
LIN {X 0,Y 539.121,Z 387.075,A -85,B 0,C 180,E1 -4029.671,E2 -4029.671} C_VEL
LIN {X 0,Y 538.856,Z 396.809,A -85,B 0,C 180,E1 -4031.147,E2 -4031.147} C_VEL
LIN {X 0,Y 541.026,Z 407.878,A -85,B 0,C 180,E1 -4031.387,E2 -4031.387} C_VEL
LIN {X 0,Y 540.797,Z 423.45,A -85,B 0,C 180,E1 -4031.711,E2 -4031.711} C_VEL
LIN {X 0,Y 540.555,Z 438.338,A -85,B 0,C 180,E1 -4032.177,E2 -4032.177} C_VEL
LIN {X 0,Y 540.192,Z 452.813,A -85,B 0,C 180,E1 -4032.784,E2 -4032.784} C_VEL
LIN {X 0,Y 539.777,Z 467.095,A -85,B 0,C 180,E1 -4033.549,E2 -4033.549} C_VEL
LIN {X 0,Y 539.392,Z 480.962,A -85,B 0,C 180,E1 -4034.477,E2 -4034.477} C_VEL
LIN {X 0,Y 538.979,Z 493.154,A -85,B 0,C 180,E1 -4035.463,E2 -4035.463} C_VEL
LIN {X 0,Y 538.612,Z 504.968,A -85,B 0,C 180,E1 -4036.608,E2 -4036.608} C_VEL
LIN {X 0,Y 538.305,Z 514.907,A -85,B 0,C 180,E1 -4037.751,E2 -4037.751} C_VEL
LIN {X 0,Y 538.111,Z 524.626,A -85,B 0,C 180,E1 -4039.084,E2 -4039.084} C_VEL
LIN {X 0,Y 537.824,Z 532.727,A -85,B 0,C 180,E1 -4040.409,E2 -4040.409} C_VEL
LIN {X 0,Y 537.734,Z 539.422,A -85,B 0,C 180,E1 -4041.734,E2 -4041.734} C_VEL
LIN {X 0,Y 537.618,Z 545.605,A -85,B 0,C 180,E1 -4043.244,E2 -4043.244} C_VEL
LIN {X 0,Y 537.574,Z 550.385,A -85,B 0,C 180,E1 -4044.749,E2 -4044.749} C_VEL
LIN {X 0,Y 537.561,Z 553.888,A -85,B 0,C 180,E1 -4046.252,E2 -4046.252} C_VEL
LIN {X 0,Y 537.488,Z 556.191,A -85,B 0,C 180,E1 -4047.752,E2 -4047.752} C_VEL
LIN {X 0,Y 537.44,Z 557.348,A -85,B 0,C 180,E1 -4049.251,E2 -4049.251} C_VEL
LIN {X 0,Y 537.44,Z 557.347,A -85,B 0,C 180,E1 -4050.749,E2 -4050.749} C_VEL
LIN {X 0,Y 537.488,Z 556.187,A -85,B 0,C 180,E1 -4052.248,E2 -4052.248} C_VEL
LIN {X 0,Y 537.561,Z 553.884,A -85,B 0,C 180,E1 -4053.748,E2 -4053.748} C_VEL
LIN {X 0,Y 537.574,Z 550.386,A -85,B 0,C 180,E1 -4055.251,E2 -4055.251} C_VEL
LIN {X 0,Y 537.664,Z 545.608,A -85,B 0,C 180,E1 -4056.756,E2 -4056.756} C_VEL
LIN {X 0,Y 537.734,Z 539.42,A -85,B 0,C 180,E1 -4058.266,E2 -4058.266} C_VEL
LIN {X 0,Y 537.859,Z 531.643,A -85,B 0,C 180,E1 -4059.78,E2 -4059.78} C_VEL
LIN {X 0,Y 538.102,Z 523.366,A -85,B 0,C 180,E1 -4061.107,E2 -4061.107} C_VEL
LIN {X 0,Y 538.358,Z 513.39,A -85,B 0,C 180,E1 -4062.439,E2 -4062.439} C_VEL
LIN {X 0,Y 538.662,Z 503.183,A -85,B 0,C 180,E1 -4063.583,E2 -4063.583} C_VEL
LIN {X 0,Y 539.022,Z 491.016,A -85,B 0,C 180,E1 -4064.729,E2 -4064.729} C_VEL
LIN {X 0,Y 539.474,Z 478.823,A -85,B 0,C 180,E1 -4065.682,E2 -4065.682} C_VEL
LIN {X 0,Y 539.847,Z 465.502,A -85,B 0,C 180,E1 -4066.546,E2 -4066.546} C_VEL
LIN {X 0,Y 540.232,Z 450.817,A -85,B 0,C 180,E1 -4067.313,E2 -4067.313} C_VEL
LIN {X 0,Y 540.598,Z 435.856,A -85,B 0,C 180,E1 -4067.915,E2 -4067.915} C_VEL
LIN {X 0,Y 540.882,Z 420.208,A -85,B 0,C 180,E1 -4068.373,E2 -4068.373} C_VEL
LIN {X 0,Y 540.877,Z 406.75,A -85,B 0,C 180,E1 -4068.636,E2 -4068.636} C_VEL
LIN {X 0,Y 538.87,Z 396.784,A -85,B 0,C 180,E1 -4068.856,E2 -4068.856} C_VEL
LIN {X 0,Y 539.131,Z 382.404,A -85,B 0,C 180,E1 -4071.007,E2 -4071.007} C_VEL
LIN {X 0,Y 539.418,Z 364.604,A -85,B 0,C 180,E1 -4073.618,E2 -4073.618} C_VEL
LIN {X 0,Y 539.785,Z 344.831,A -85,B 0,C 180,E1 -4076.692,E2 -4076.692} C_VEL
LIN {X 0,Y 540.199,Z 330.22,A -85,B 0,C 180,E1 -4079.065,E2 -4079.065} C_VEL
LIN {X 0,Y 540.804,Z 316.173,A -85,B 0,C 180,E1 -4081.538,E2 -4081.538} C_VEL
LIN {X 0,Y 541.8,Z 304.067,A -85,B 0,C 180,E1 -4083.903,E2 -4083.903} C_VEL
LIN {X 0,Y 542.06,Z 300.052,A -85,B 0,C 180,E1 -4084.784,E2 -4084.784} C_VEL
LIN {X 0,Y 540.756,Z 294.429,A -85,B 0,C 180,E1 -4086.313,E2 -4086.313} C_VEL
LIN {X 0,Y 538.978,Z 287.887,A -85,B 0,C 180,E1 -4088.522,E2 -4088.522} C_VEL
LIN {X 0,Y 538.043,Z 284.093,A -85,B 0,C 180,E1 -4090.254,E2 -4090.254} C_VEL
LIN {X 0,Y 538.028,Z 284.095,A -85,B 0,C 180,E1 -4092.988,E2 -4092.988} C_VEL
LIN {X 0,Y 538.005,Z 284.097,A -85,B 0,C 180,E1 -4096.184,E2 -4096.184} C_VEL
LIN {X 0,Y 538.05,Z 284.092,A -85,B 0,C 180,E1 -4099.253,E2 -4099.253} C_VEL
LIN {X 0,Y 537.994,Z 284.099,A -85,B 0,C 180,E1 -4102.122,E2 -4102.122} C_VEL
LIN {X 0,Y 538.247,Z 285.908,A -85,B 0,C 180,E1 -4104.052,E2 -4104.052} C_VEL
LIN {X 0,Y 538.288,Z 288.606,A -85,B 0,C 180,E1 -4106.745,E2 -4106.745} C_VEL
LIN {X 0,Y 538.188,Z 291.281,A -85,B 0,C 180,E1 -4109.528,E2 -4109.528} C_VEL
LIN {X 0,Y 538.154,Z 293.471,A -85,B 0,C 180,E1 -4111.957,E2 -4111.957} C_VEL
LIN {X 0,Y 538.111,Z 295.627,A -85,B 0,C 180,E1 -4114.469,E2 -4114.469} C_VEL
LIN {X 0,Y 538.004,Z 297.753,A -85,B 0,C 180,E1 -4116.928,E2 -4116.928} C_VEL
LIN {X 0,Y 537.89,Z 300.514,A -85,B 0,C 180,E1 -4120.178,E2 -4120.178} C_VEL
LIN {X 0,Y 537.811,Z 302.553,A -85,B 0,C 180,E1 -4122.545,E2 -4122.545} C_VEL
LIN {X 0,Y 537.705,Z 305.13,A -85,B 0,C 180,E1 -4125.621,E2 -4125.621} C_VEL
LIN {X 0,Y 537.678,Z 306.142,A -85,B 0,C 180,E1 -4126.705,E2 -4126.705} C_VEL
LIN {X 0,Y 539.391,Z 314.562,A -85,B 0,C 180,E1 -4126.975,E2 -4126.975} C_VEL
LIN {X 0,Y 539.176,Z 326.659,A -85,B 0,C 180,E1 -4127.389,E2 -4127.389} C_VEL
LIN {X 0,Y 538.963,Z 338.675,A -85,B 0,C 180,E1 -4127.958,E2 -4127.958} C_VEL
LIN {X 0,Y 538.71,Z 350.917,A -85,B 0,C 180,E1 -4128.715,E2 -4128.715} C_VEL
LIN {X 0,Y 538.444,Z 361.692,A -85,B 0,C 180,E1 -4129.566,E2 -4129.566} C_VEL
LIN {X 0,Y 538.206,Z 372.167,A -85,B 0,C 180,E1 -4130.606,E2 -4130.606} C_VEL
LIN {X 0,Y 538.019,Z 379.892,A -85,B 0,C 180,E1 -4131.55,E2 -4131.55} C_VEL
LIN {X 0,Y 537.822,Z 387.445,A -85,B 0,C 180,E1 -4132.68,E2 -4132.68} C_VEL
LIN {X 0,Y 537.717,Z 394.35,A -85,B 0,C 180,E1 -4133.998,E2 -4133.998} C_VEL
LIN {X 0,Y 537.547,Z 398.967,A -85,B 0,C 180,E1 -4135.125,E2 -4135.125} C_VEL
LIN {X 0,Y 537.591,Z 402.469,A -85,B 0,C 180,E1 -4136.252,E2 -4136.252} C_VEL
LIN {X 0,Y 537.58,Z 404.282,A -85,B 0,C 180,E1 -4137.003,E2 -4137.003} C_VEL
LIN {X 0,Y 537.489,Z 405.667,A -85,B 0,C 180,E1 -4137.752,E2 -4137.752} C_VEL
LIN {X 0,Y 537.443,Z 407.256,A -85,B 0,C 180,E1 -4139.251,E2 -4139.251} C_VEL
LIN {X 0,Y 537.442,Z 407.496,A -85,B 0,C 180,E1 -4140,E2 -4140} C_VEL
LIN {X 0,Y 537.442,Z 407.314,A -85,B 0,C 180,E1 -4140.749,E2 -4140.749} C_VEL
LIN {X 0,Y 537.489,Z 405.782,A -85,B 0,C 180,E1 -4142.248,E2 -4142.248} C_VEL
LIN {X 0,Y 537.552,Z 404.447,A -85,B 0,C 180,E1 -4142.998,E2 -4142.998} C_VEL
LIN {X 0,Y 537.603,Z 401.637,A -85,B 0,C 180,E1 -4144.123,E2 -4144.123} C_VEL
LIN {X 0,Y 537.587,Z 397.834,A -85,B 0,C 180,E1 -4145.251,E2 -4145.251} C_VEL
LIN {X 0,Y 537.683,Z 393.182,A -85,B 0,C 180,E1 -4146.32,E2 -4146.32} C_VEL
LIN {X 0,Y 537.806,Z 386.678,A -85,B 0,C 180,E1 -4147.509,E2 -4147.509} C_VEL
LIN {X 0,Y 537.988,Z 378.878,A -85,B 0,C 180,E1 -4148.64,E2 -4148.64} C_VEL
LIN {X 0,Y 538.167,Z 370.913,A -85,B 0,C 180,E1 -4149.585,E2 -4149.585} C_VEL
LIN {X 0,Y 538.435,Z 361.17,A -85,B 0,C 180,E1 -4150.529,E2 -4150.529} C_VEL
LIN {X 0,Y 538.641,Z 351.591,A -85,B 0,C 180,E1 -4151.287,E2 -4151.287} C_VEL
LIN {X 0,Y 538.827,Z 340.828,A -85,B 0,C 180,E1 -4151.974,E2 -4151.974} C_VEL
LIN {X 0,Y 539.041,Z 328.827,A -85,B 0,C 180,E1 -4152.566,E2 -4152.566} C_VEL
LIN {X 0,Y 539.267,Z 315.763,A -85,B 0,C 180,E1 -4153.04,E2 -4153.04} C_VEL
LIN {X 0,Y 538.23,Z 308.43,A -85,B 0,C 180,E1 -4153.263,E2 -4153.263} C_VEL
LIN {X 0,Y 537.539,Z 305.146,A -85,B 0,C 180,E1 -4153.371,E2 -4153.371} C_VEL
LIN {X 0,Y 537.566,Z 302.546,A -85,B 0,C 180,E1 -4155.935,E2 -4155.935} C_VEL
LIN {X 0,Y 537.574,Z 300.14,A -85,B 0,C 180,E1 -4158.286,E2 -4158.286} C_VEL
LIN {X 0,Y 537.628,Z 297.549,A -85,B 0,C 180,E1 -4160.668,E2 -4160.668} C_VEL
LIN {X 0,Y 537.665,Z 294.143,A -85,B 0,C 180,E1 -4163.904,E2 -4163.904} C_VEL
LIN {X 0,Y 537.685,Z 291.484,A -85,B 0,C 180,E1 -4166.386,E2 -4166.386} C_VEL
LIN {X 0,Y 537.746,Z 288.826,A -85,B 0,C 180,E1 -4168.919,E2 -4168.919} C_VEL
LIN {X 0,Y 537.693,Z 285.59,A -85,B 0,C 180,E1 -4171.832,E2 -4171.832} C_VEL
LIN {X 0,Y 537.731,Z 284.132,A -85,B 0,C 180,E1 -4173.294,E2 -4173.294} C_VEL
LIN {X 0,Y 537.95,Z 284.098,A -85,B 0,C 180,E1 -4175.904,E2 -4175.904} C_VEL
LIN {X 0,Y 537.962,Z 284.096,A -85,B 0,C 180,E1 -4176.308,E2 -4176.308} C_VEL
LIN {X 0,Y 537.33,Z 284.181,A -85,B 0,C 180,E1 -4176.933,E2 -4176.933} C_VEL
LIN {X 0,Y 534.511,Z 284.529,A -85,B 0,C 180,E1 -4177.949,E2 -4177.949} C_VEL
LIN {X 0,Y 532.109,Z 284.83,A -85,B 0,C 180,E1 -4178.766,E2 -4178.766} C_VEL
LIN {X 0,Y 531.072,Z 284.956,A -85,B 0,C 180,E1 -4179.398,E2 -4179.398} C_VEL
LIN {X 0,Y 530.985,Z 284.965,A -85,B 0,C 180,E1 -4179.611,E2 -4179.611} C_VEL
LIN {X 0,Y 530.981,Z 284.97,A -85,B 0,C 180,E1 -4182.457,E2 -4182.457} C_VEL
LIN {X 0,Y 530.973,Z 284.968,A -85,B 0,C 180,E1 -4185.623,E2 -4185.623} C_VEL
LIN {X 0,Y 530.917,Z 284.978,A -85,B 0,C 180,E1 -4188.557,E2 -4188.557} C_VEL
LIN {X 0,Y 530.861,Z 284.987,A -85,B 0,C 180,E1 -4189.556,E2 -4189.556} C_VEL
LIN {X 0,Y 530.919,Z 287.912,A -85,B 0,C 180,E1 -4191.526,E2 -4191.526} C_VEL
LIN {X 0,Y 530.852,Z 292.143,A -85,B 0,C 180,E1 -4194.372,E2 -4194.372} C_VEL
LIN {X 0,Y 530.839,Z 296.004,A -85,B 0,C 180,E1 -4197.124,E2 -4197.124} C_VEL
LIN {X 0,Y 530.757,Z 299.627,A -85,B 0,C 180,E1 -4199.789,E2 -4199.789} C_VEL
LIN {X 0,Y 530.714,Z 303.467,A -85,B 0,C 180,E1 -4202.53,E2 -4202.53} C_VEL
LIN {X 0,Y 530.671,Z 306.931,A -85,B 0,C 180,E1 -4204.925,E2 -4204.925} C_VEL
LIN {X 0,Y 530.646,Z 311.336,A -85,B 0,C 180,E1 -4207.987,E2 -4207.987} C_VEL
LIN {X 0,Y 530.584,Z 315.503,A -85,B 0,C 180,E1 -4210.966,E2 -4210.966} C_VEL
LIN {X 0,Y 531.26,Z 317.888,A -85,B 0,C 180,E1 -4211.059,E2 -4211.059} C_VEL
LIN {X 0,Y 534.213,Z 329.904,A -85,B 0,C 180,E1 -4211.415,E2 -4211.415} C_VEL
LIN {X 0,Y 533.947,Z 344.732,A -85,B 0,C 180,E1 -4211.841,E2 -4211.841} C_VEL
LIN {X 0,Y 533.507,Z 359.278,A -85,B 0,C 180,E1 -4212.412,E2 -4212.412} C_VEL
LIN {X 0,Y 533.129,Z 373.493,A -85,B 0,C 180,E1 -4213.141,E2 -4213.141} C_VEL
LIN {X 0,Y 532.693,Z 385.68,A -85,B 0,C 180,E1 -4213.915,E2 -4213.915} C_VEL
LIN {X 0,Y 532.297,Z 397.107,A -85,B 0,C 180,E1 -4214.787,E2 -4214.787} C_VEL
LIN {X 0,Y 531.944,Z 406.831,A -85,B 0,C 180,E1 -4215.657,E2 -4215.657} C_VEL
LIN {X 0,Y 531.606,Z 416.265,A -85,B 0,C 180,E1 -4216.623,E2 -4216.623} C_VEL
LIN {X 0,Y 531.297,Z 424.475,A -85,B 0,C 180,E1 -4217.587,E2 -4217.587} C_VEL
LIN {X 0,Y 531.057,Z 432.99,A -85,B 0,C 180,E1 -4218.743,E2 -4218.743} C_VEL
LIN {X 0,Y 530.816,Z 441.412,A -85,B 0,C 180,E1 -4220.089,E2 -4220.089} C_VEL
LIN {X 0,Y 530.667,Z 449.164,A -85,B 0,C 180,E1 -4221.623,E2 -4221.623} C_VEL
LIN {X 0,Y 530.573,Z 453.986,A -85,B 0,C 180,E1 -4222.771,E2 -4222.771} C_VEL
LIN {X 0,Y 530.516,Z 458.008,A -85,B 0,C 180,E1 -4223.916,E2 -4223.916} C_VEL
LIN {X 0,Y 530.412,Z 462.145,A -85,B 0,C 180,E1 -4225.44,E2 -4225.44} C_VEL
LIN {X 0,Y 530.481,Z 463.832,A -85,B 0,C 180,E1 -4226.202,E2 -4226.202} C_VEL
LIN {X 0,Y 530.409,Z 466.127,A -85,B 0,C 180,E1 -4227.722,E2 -4227.722} C_VEL
LIN {X 0,Y 530.34,Z 467.271,A -85,B 0,C 180,E1 -4229.241,E2 -4229.241} C_VEL
LIN {X 0,Y 530.341,Z 467.496,A -85,B 0,C 180,E1 -4230,E2 -4230} C_VEL
LIN {X 0,Y 530.36,Z 466.944,A -85,B 0,C 180,E1 -4231.519,E2 -4231.519} C_VEL
LIN {X 0,Y 530.45,Z 465.227,A -85,B 0,C 180,E1 -4233.038,E2 -4233.038} C_VEL
LIN {X 0,Y 530.481,Z 464,A -85,B 0,C 180,E1 -4233.798,E2 -4233.798} C_VEL
LIN {X 0,Y 530.544,Z 459.402,A -85,B 0,C 180,E1 -4235.702,E2 -4235.702} C_VEL
